C07264=1053.919,247.407,-97.139,172.328,35.943,156.751
C07265=1053.925,247.656,-97.168,172.330,35.946,156.752
C07266=1053.932,247.903,-97.196,172.333,35.950,156.753
C07267=1053.938,248.152,-97.225,172.335,35.954,156.754
C07268=1053.944,248.400,-97.254,172.337,35.957,156.754
C07269=1053.950,248.641,-97.282,172.340,35.960,156.755
C07270=1053.956,248.882,-97.309,172.343,35.964,156.756
C07271=1053.961,249.122,-97.337,172.345,35.967,156.757
C07272=1053.968,249.364,-97.365,172.348,35.970,156.757
C07273=1053.974,249.605,-97.393,172.350,35.974,156.758
C07274=1053.980,249.845,-97.421,172.353,35.977,156.759
C07275=1053.986,250.087,-97.448,172.355,35.980,156.759
C07276=1053.992,250.327,-97.476,172.357,35.984,156.760
C07277=1053.999,250.575,-97.505,172.360,35.987,156.761
C07278=1054.005,250.824,-97.533,172.362,35.991,156.761
C07279=1054.011,251.072,-97.563,172.364,35.994,156.762
C07280=1054.017,251.320,-97.592,172.367,35.998,156.763
C07281=1054.023,251.569,-97.620,172.369,36.001,156.764
C07282=1054.029,251.817,-97.649,172.372,36.005,156.764
C07283=1054.036,252.065,-97.678,172.374,36.008,156.765
C07284=1054.043,252.313,-97.706,172.377,36.012,156.766
C07285=1054.049,252.561,-97.735,172.380,36.015,156.766
C07286=1054.055,252.810,-97.764,172.382,36.018,156.767
C07287=1054.061,253.058,-97.793,172.384,36.022,156.768
C07288=1054.067,253.306,-97.822,172.387,36.025,156.769
C07289=1054.074,253.554,-97.851,172.389,36.029,156.769
C07290=1054.080,253.803,-97.880,172.392,36.033,156.770
C07291=1054.086,254.052,-97.909,172.395,36.036,156.771
C07292=1054.093,254.300,-97.938,172.397,36.039,156.771
C07293=1054.100,254.548,-97.966,172.400,36.043,156.772
C07294=1054.106,254.796,-97.995,172.402,36.046,156.773
C07295=1054.112,255.044,-98.024,172.404,36.050,156.774
C07296=1054.118,255.292,-98.053,172.407,36.053,156.774
C07297=1054.125,255.540,-98.082,172.410,36.056,156.775
C07298=1054.131,255.789,-98.111,172.413,36.060,156.776
C07299=1054.138,256.037,-98.141,172.415,36.063,156.777
C07300=1054.144,256.286,-98.170,172.417,36.066,156.777
C07301=1054.150,256.534,-98.199,172.420,36.070,156.778
C07302=1054.156,256.782,-98.228,172.423,36.073,156.779
C07303=1054.163,257.030,-98.257,172.425,36.077,156.779
C07304=1054.169,257.278,-98.286,172.428,36.081,156.780
C07305=1054.176,257.527,-98.315,172.430,36.083,156.781
C07306=1054.183,257.775,-98.344,172.433,36.087,156.782
C07307=1054.189,258.023,-98.373,172.436,36.091,156.782
C07308=1054.195,258.271,-98.402,172.438,36.094,156.783
C07309=1054.201,258.519,-98.431,172.441,36.097,156.784
C07310=1054.208,258.768,-98.460,172.443,36.101,156.784
C07311=1054.215,259.016,-98.489,172.445,36.104,156.785
C07312=1054.221,259.264,-98.518,172.449,36.108,156.786
C07313=1054.227,259.512,-98.547,172.451,36.111,156.787
C07314=1054.234,259.761,-98.577,172.454,36.114,156.787
C07315=1054.241,260.009,-98.607,172.456,36.118,156.788
C07316=1054.247,260.257,-98.636,172.459,36.121,156.789
C07317=1054.253,260.505,-98.665,172.462,36.124,156.789
C07318=1054.260,260.754,-98.694,172.464,36.128,156.790
C07319=1054.266,261.002,-98.723,172.467,36.131,156.791
C07320=1054.273,261.249,-98.753,172.470,36.135,156.792
C07321=1054.279,261.498,-98.782,172.472,36.138,156.792
C07322=1054.286,261.746,-98.811,172.475,36.141,156.793
C07323=1054.292,261.995,-98.840,172.477,36.145,156.794
C07324=1054.298,262.243,-98.869,172.481,36.149,156.794
C07325=1054.304,262.456,-98.895,172.483,36.151,156.795
C07326=1054.310,262.670,-98.921,172.485,36.154,156.796
C07327=1054.316,262.884,-98.945,172.487,36.157,156.796
C07328=1054.321,263.098,-98.971,172.490,36.160,156.797
C07329=1054.327,263.312,-98.997,172.491,36.163,156.798
C07330=1054.332,263.525,-99.022,172.494,36.166,156.798
C07331=1054.337,263.740,-99.048,172.496,36.169,156.799
C07332=1054.343,263.953,-99.073,172.498,36.172,156.799
C07333=1054.351,264.254,-99.110,172.502,36.176,156.800
C07334=1054.358,264.554,-99.145,172.505,36.180,156.801
C07335=1054.366,264.855,-99.181,172.509,36.185,156.802
C07336=1054.373,265.155,-99.217,172.511,36.189,156.803
C07337=1054.380,265.403,-99.247,172.515,36.192,156.804
C07338=1054.386,265.651,-99.276,172.517,36.196,156.804
C07339=1054.392,265.899,-99.306,172.519,36.199,156.805
C07340=1054.399,266.148,-99.336,172.522,36.203,156.806
C07341=1054.406,266.396,-99.365,172.525,36.206,156.807
C07342=1054.411,266.644,-99.395,172.528,36.210,156.807
C07343=1054.418,266.892,-99.425,172.530,36.213,156.808
C07344=1054.424,267.140,-99.454,172.533,36.216,156.809
C07345=1054.431,267.389,-99.485,172.536,36.220,156.810
C07346=1054.437,267.636,-99.515,172.538,36.223,156.810
C07347=1054.444,267.885,-99.544,172.542,36.227,156.811
C07348=1054.450,268.133,-99.574,172.544,36.230,156.812
C07349=1054.456,268.381,-99.604,172.546,36.234,156.813
C07350=1054.462,268.629,-99.634,172.550,36.238,156.813
C07351=1054.469,268.877,-99.664,172.552,36.241,156.814
C07352=1054.475,269.126,-99.694,172.555,36.245,156.815
C07353=1054.482,269.374,-99.724,172.558,36.248,156.816
C07354=1054.488,269.622,-99.754,172.560,36.251,156.816
C07355=1054.494,269.869,-99.784,172.563,36.255,156.817
C07356=1054.500,270.118,-99.814,172.566,36.258,156.818
C07357=1054.507,270.366,-99.844,172.569,36.262,156.818
C07358=1054.513,270.614,-99.874,172.571,36.265,156.819
C07359=1054.520,270.862,-99.904,172.575,36.269,156.820
C07360=1054.526,271.110,-99.935,172.577,36.272,156.821
C07361=1054.533,271.359,-99.964,172.579,36.276,156.821
C07362=1054.539,271.606,-99.994,172.583,36.279,156.822
C07363=1054.546,271.855,-100.024,172.585,36.283,156.823
C07364=1054.551,272.102,-100.055,172.588,36.286,156.824
C07365=1054.559,272.351,-100.085,172.591,36.290,156.825
C07366=1054.564,272.598,-100.115,172.594,36.293,156.825
C07367=1054.571,272.847,-100.146,172.597,36.297,156.826
C07368=1054.577,273.094,-100.176,172.599,36.300,156.827
C07369=1054.584,273.343,-100.206,172.602,36.304,156.828
C07370=1054.590,273.591,-100.235,172.605,36.307,156.828
C07371=1054.597,273.840,-100.266,172.608,36.311,156.829
C07372=1054.602,274.088,-100.296,172.610,36.314,156.830
C07373=1054.609,274.336,-100.327,172.613,36.318,156.831
C07374=1054.615,274.584,-100.357,172.616,36.322,156.831
C07375=1054.622,274.831,-100.388,172.619,36.324,156.832
C07376=1054.629,275.079,-100.418,172.622,36.328,156.833
C07377=1054.635,275.327,-100.449,172.624,36.331,156.833
C07378=1054.641,275.575,-100.479,172.628,36.335,156.834
C07379=1054.647,275.824,-100.510,172.630,36.339,156.835
C07380=1054.654,276.071,-100.540,172.633,36.342,156.836
C07381=1054.660,276.314,-100.569,172.636,36.346,156.836
C07382=1054.666,276.555,-100.599,172.638,36.349,156.837
C07383=1054.672,276.798,-100.629,172.642,36.353,156.838
C07384=1054.679,277.040,-100.659,172.644,36.356,156.839
C07385=1054.685,277.282,-100.689,172.647,36.360,156.839
C07386=1054.691,277.524,-100.719,172.650,36.363,156.840
C07387=1054.697,277.766,-100.748,172.652,36.367,156.841
C07388=1054.703,278.007,-100.778,172.656,36.370,156.842
C07389=1054.710,278.256,-100.808,172.658,36.373,156.842
C07390=1054.716,278.504,-100.839,172.661,36.377,156.843
C07391=1054.723,278.751,-100.870,172.664,36.381,156.844
C07392=1054.729,279.000,-100.901,172.667,36.384,156.845
C07393=1054.735,279.248,-100.931,172.670,36.388,156.846
C07394=1054.742,279.496,-100.961,172.673,36.391,156.846
C07395=1054.749,279.744,-100.993,172.676,36.395,156.847
C07396=1054.755,279.992,-101.023,172.678,36.398,156.848
C07397=1054.761,280.240,-101.054,172.682,36.402,156.849
C07398=1054.767,280.487,-101.085,172.684,36.405,156.849
C07399=1054.774,280.736,-101.116,172.688,36.409,156.850
C07400=1054.780,280.984,-101.147,172.690,36.412,156.851
C07401=1054.786,281.232,-101.178,172.693,36.416,156.852
C07402=1054.793,281.480,-101.209,172.696,36.419,156.852
C07403=1054.799,281.728,-101.240,172.699,36.423,156.853
C07404=1054.805,281.975,-101.271,172.702,36.427,156.854
C07405=1054.812,282.224,-101.301,172.704,36.430,156.855
C07406=1054.818,282.472,-101.333,172.708,36.434,156.856
C07407=1054.824,282.720,-101.363,172.710,36.437,156.856
C07408=1054.831,282.967,-101.395,172.714,36.441,156.857
C07409=1054.837,283.216,-101.425,172.716,36.444,156.858
C07410=1054.844,283.463,-101.456,172.720,36.448,156.859
C07411=1054.850,283.712,-101.487,172.722,36.452,156.859
C07412=1054.857,283.960,-101.519,172.726,36.455,156.860
C07413=1054.863,284.207,-101.549,172.728,36.459,156.861
C07414=1054.869,284.455,-101.580,172.732,36.462,156.862
C07415=1054.876,284.703,-101.612,172.734,36.466,156.862
C07416=1054.882,284.952,-101.643,172.737,36.469,156.863
C07417=1054.889,285.199,-101.674,172.740,36.473,156.864
C07418=1054.895,285.447,-101.705,172.743,36.477,156.865
C07419=1054.902,285.695,-101.736,172.746,36.481,156.866
C07420=1054.908,285.944,-101.768,172.749,36.484,156.866
C07421=1054.914,286.191,-101.799,172.753,36.488,156.867
C07422=1054.920,286.439,-101.830,172.755,36.491,156.868
C07423=1054.927,286.687,-101.861,172.759,36.495,156.869
C07424=1054.934,286.935,-101.892,172.761,36.498,156.869
C07425=1054.940,287.183,-101.924,172.765,36.502,156.870
C07426=1054.946,287.431,-101.954,172.767,36.506,156.871
C07427=1054.953,287.679,-101.986,172.771,36.509,156.872
C07428=1054.960,287.927,-102.017,172.773,36.513,156.873
C07429=1054.966,288.175,-102.049,172.776,36.516,156.873
C07430=1054.973,288.422,-102.080,172.780,36.520,156.874
C07431=1054.978,288.670,-102.112,172.782,36.524,156.875
C07432=1054.985,288.918,-102.143,172.786,36.527,156.876
C07433=1054.992,289.166,-102.174,172.788,36.531,156.877
C07434=1054.998,289.414,-102.205,172.792,36.534,156.877
C07435=1055.004,289.662,-102.237,172.794,36.538,156.878
C07436=1055.011,289.910,-102.269,172.798,36.542,156.879
C07437=1055.017,290.158,-102.300,172.801,36.545,156.880
C07438=1055.024,290.405,-102.332,172.804,36.549,156.881
C07439=1055.030,290.652,-102.363,172.807,36.553,156.881
C07440=1055.037,290.900,-102.394,172.810,36.556,156.882
C07441=1055.042,291.147,-102.426,172.813,36.560,156.883
C07442=1055.049,291.395,-102.458,172.817,36.563,156.884
C07443=1055.056,291.643,-102.490,172.819,36.567,156.885
C07444=1055.062,291.890,-102.521,172.823,36.571,156.885
C07445=1055.068,292.138,-102.553,172.825,36.574,156.886
C07446=1055.075,292.386,-102.584,172.829,36.578,156.887
C07447=1055.082,292.634,-102.616,172.832,36.582,156.888
C07448=1055.088,292.882,-102.648,172.835,36.585,156.889
C07449=1055.095,293.129,-102.680,172.838,36.589,156.889
C07450=1055.101,293.377,-102.711,172.842,36.593,156.890
C07451=1055.107,293.625,-102.743,172.844,36.596,156.891
C07452=1055.114,293.873,-102.775,172.848,36.600,156.892
C07453=1055.120,294.121,-102.806,172.850,36.604,156.893
C07454=1055.127,294.368,-102.838,172.854,36.607,156.893
C07455=1055.133,294.616,-102.870,172.857,36.611,156.894
C07456=1055.139,294.864,-102.902,172.860,36.615,156.895
C07457=1055.146,295.112,-102.933,172.863,36.618,156.896
C07458=1055.152,295.360,-102.966,172.867,36.622,156.897
C07459=1055.159,295.608,-102.998,172.869,36.626,156.898
C07460=1055.165,295.856,-103.030,172.872,36.629,156.898
C07461=1055.172,296.103,-103.062,172.876,36.633,156.899
C07462=1055.178,296.351,-103.094,172.879,36.637,156.900
C07463=1055.185,296.599,-103.126,172.882,36.640,156.901
C07464=1055.191,296.847,-103.158,172.886,36.644,156.902
C07465=1055.197,297.095,-103.190,172.888,36.648,156.903
C07466=1055.204,297.342,-103.222,172.892,36.652,156.903
C07467=1055.210,297.591,-103.254,172.895,36.656,156.904
C07468=1055.216,297.838,-103.287,172.898,36.659,156.905
C07469=1055.222,298.086,-103.319,172.901,36.663,156.906
C07470=1055.229,298.334,-103.352,172.905,36.667,156.907
C07471=1055.236,298.581,-103.384,172.907,36.671,156.908
C07472=1055.242,298.829,-103.416,172.911,36.674,156.908
C07473=1055.248,299.077,-103.449,172.914,36.678,156.909
C07474=1055.254,299.325,-103.481,172.917,36.682,156.910
C07475=1055.261,299.573,-103.513,172.920,36.686,156.911
C07476=1055.267,299.820,-103.545,172.924,36.690,156.912
C07477=1055.273,300.068,-103.577,172.926,36.693,156.913
C07478=1055.280,300.316,-103.610,172.930,36.697,156.913
C07479=1055.286,300.564,-103.643,172.933,36.701,156.914
C07480=1055.293,300.811,-103.674,172.937,36.705,156.915
C07481=1055.299,301.059,-103.707,172.939,36.709,156.916
C07482=1055.305,301.307,-103.740,172.943,36.712,156.917
C07483=1055.311,301.555,-103.772,172.946,36.717,156.918
C07484=1055.317,301.802,-103.805,172.950,36.720,156.918
C07485=1055.324,302.050,-103.837,172.953,36.724,156.919
C07486=1055.331,302.298,-103.870,172.956,36.728,156.920
C07487=1055.338,302.546,-103.903,172.960,36.731,156.921
C07488=1055.344,302.794,-103.935,172.963,36.736,156.922
C07489=1055.350,303.041,-103.967,172.966,36.739,156.923
C07490=1055.356,303.289,-104.000,172.969,36.743,156.924
C07491=1055.363,303.537,-104.033,172.973,36.747,156.924
C07492=1055.370,303.784,-104.065,172.976,36.751,156.925
C07493=1055.376,304.047,-104.100,172.979,36.755,156.926
C07494=1055.383,304.310,-104.134,172.982,36.759,156.927
C07495=1055.390,304.573,-104.169,172.986,36.763,156.928
C07496=1055.396,304.836,-104.204,172.990,36.767,156.929
C07497=1055.404,305.084,-104.236,172.993,36.771,156.930
C07498=1055.410,305.332,-104.269,172.997,36.775,156.931
C07499=1055.417,305.580,-104.302,173.000,36.778,156.931
C07500=1055.423,305.827,-104.334,173.004,36.782,156.932
C07501=1055.429,306.075,-104.367,173.006,36.786,156.933
C07502=1055.436,306.323,-104.400,173.010,36.790,156.934
C07503=1055.442,306.571,-104.433,173.013,36.794,156.935
C07504=1055.449,306.818,-104.466,173.017,36.798,156.936
C07505=1055.456,307.065,-104.499,173.020,36.801,156.937
C07506=1055.463,307.313,-104.532,173.023,36.805,156.938
C07507=1055.469,307.561,-104.564,173.027,36.809,156.938
C07508=1055.475,307.808,-104.597,173.030,36.813,156.939
C07509=1055.482,308.057,-104.630,173.034,36.817,156.940
C07510=1055.489,308.304,-104.663,173.037,36.821,156.941
C07511=1055.495,308.552,-104.696,173.041,36.825,156.942
C07512=1055.502,308.800,-104.729,173.044,36.828,156.943
C07513=1055.508,309.047,-104.762,173.047,36.832,156.944
C07514=1055.515,309.294,-104.795,173.051,36.836,156.945
C07515=1055.522,309.543,-104.828,173.054,36.840,156.945
C07516=1055.529,309.790,-104.860,173.058,36.844,156.946
C07517=1055.535,310.037,-104.894,173.061,36.848,156.947
C07518=1055.542,310.286,-104.927,173.065,36.852,156.948
C07519=1055.548,310.533,-104.960,173.068,36.855,156.949
C07520=1055.555,310.781,-104.993,173.071,36.859,156.950
C07521=1055.562,311.028,-105.026,173.074,36.863,156.951
C07522=1055.569,311.277,-105.059,173.078,36.867,156.952
C07523=1055.575,311.524,-105.092,173.082,36.871,156.952
C07524=1055.582,311.771,-105.126,173.085,36.875,156.953
C07525=1055.589,312.020,-105.159,173.089,36.879,156.954
C07526=1055.595,312.267,-105.192,173.092,36.883,156.955
C07527=1055.602,312.515,-105.225,173.096,36.886,156.956
C07528=1055.608,312.762,-105.258,173.099,36.890,156.957
C07529=1055.616,313.010,-105.292,173.103,36.894,156.958
C07530=1055.622,313.258,-105.325,173.107,36.898,156.959
C07531=1055.629,313.505,-105.358,173.109,36.902,156.959
C07532=1055.635,313.753,-105.391,173.113,36.906,156.960
C07533=1055.642,314.001,-105.426,173.116,36.910,156.961
C07534=1055.648,314.248,-105.459,173.120,36.914,156.962
C07535=1055.655,314.497,-105.493,173.124,36.918,156.963
C07536=1055.661,314.743,-105.526,173.127,36.922,156.964
C07537=1055.667,314.991,-105.560,173.131,36.926,156.965
C07538=1055.674,315.239,-105.593,173.134,36.930,156.966
C07539=1055.681,315.486,-105.627,173.138,36.934,156.967
C07540=1055.687,315.734,-105.661,173.142,36.939,156.968
C07541=1055.693,315.982,-105.694,173.144,36.943,156.969
C07542=1055.700,316.230,-105.728,173.148,36.947,156.970
C07543=1055.706,316.477,-105.762,173.151,36.951,156.970
C07544=1055.713,316.725,-105.796,173.155,36.955,156.971
C07545=1055.719,316.972,-105.829,173.159,36.959,156.972
C07546=1055.726,317.220,-105.863,173.162,36.963,156.973
C07547=1055.732,317.467,-105.897,173.166,36.967,156.974
C07548=1055.739,317.715,-105.931,173.170,36.971,156.975
C07549=1055.745,317.982,-105.968,173.173,36.975,156.976
C07550=1055.752,318.249,-106.004,173.177,36.980,156.977
C07551=1055.759,318.516,-106.041,173.182,36.984,156.978
C07552=1055.767,318.784,-106.078,173.185,36.989,156.979
C07553=1055.773,319.031,-106.111,173.189,36.993,156.980
C07554=1055.780,319.279,-106.146,173.192,36.997,156.981
C07555=1055.786,319.527,-106.179,173.196,37.001,156.982
C07556=1055.792,319.774,-106.213,173.200,37.005,156.983
C07557=1055.800,320.022,-106.247,173.203,37.009,156.984
C07558=1055.805,320.269,-106.281,173.207,37.013,156.985
C07559=1055.813,320.517,-106.315,173.211,37.017,156.986
C07560=1055.819,320.764,-106.350,173.214,37.021,156.987
C07561=1055.826,321.011,-106.383,173.218,37.026,156.988
C07562=1055.832,321.259,-106.418,173.221,37.030,156.989
C07563=1055.839,321.507,-106.452,173.225,37.034,156.990
C07564=1055.845,321.754,-106.486,173.229,37.038,156.990
C07565=1055.852,322.002,-106.520,173.232,37.042,156.992
C07566=1055.859,322.250,-106.554,173.236,37.046,156.992
C07567=1055.866,322.498,-106.588,173.240,37.050,156.993
C07568=1055.872,322.745,-106.622,173.243,37.054,156.994
C07569=1055.879,322.992,-106.657,173.247,37.059,156.995
C07570=1055.885,323.240,-106.691,173.251,37.063,156.996
C07571=1055.893,323.488,-106.725,173.254,37.067,156.997
C07572=1055.898,323.735,-106.759,173.258,37.071,156.998
C07573=1055.906,323.983,-106.793,173.262,37.075,156.999
C07574=1055.912,324.230,-106.828,173.265,37.079,157.000
C07575=1055.919,324.478,-106.862,173.269,37.084,157.001
C07576=1055.926,324.726,-106.896,173.272,37.088,157.002
C07577=1055.932,324.972,-106.931,173.276,37.092,157.003
C07578=1055.939,325.220,-106.965,173.280,37.096,157.004
C07579=1055.946,325.468,-106.999,173.284,37.100,157.005
C07580=1055.953,325.715,-107.034,173.288,37.105,157.006
C07581=1055.960,325.963,-107.068,173.292,37.109,157.007
C07582=1055.966,326.211,-107.103,173.295,37.113,157.008
C07583=1055.973,326.458,-107.138,173.299,37.117,157.009
C07584=1055.980,326.705,-107.171,173.303,37.121,157.010
C07585=1055.987,326.953,-107.206,173.306,37.126,157.011
C07586=1055.993,327.201,-107.241,173.310,37.130,157.012
C07587=1056.000,327.448,-107.275,173.314,37.134,157.013
C07588=1056.007,327.696,-107.310,173.318,37.138,157.014
C07589=1056.014,327.943,-107.344,173.322,37.142,157.015
C07590=1056.021,328.191,-107.379,173.326,37.147,157.016
C07591=1056.028,328.438,-107.414,173.329,37.151,157.017
C07592=1056.035,328.686,-107.448,173.333,37.155,157.018
C07593=1056.042,328.933,-107.483,173.337,37.159,157.019
C07594=1056.048,329.181,-107.518,173.341,37.164,157.020
C07595=1056.056,329.428,-107.552,173.345,37.168,157.021
C07596=1056.062,329.676,-107.587,173.349,37.172,157.022
C07597=1056.069,329.924,-107.621,173.353,37.176,157.023
C07598=1056.076,330.171,-107.657,173.356,37.181,157.024
C07599=1056.082,330.418,-107.692,173.360,37.185,157.025
C07600=1056.089,330.666,-107.727,173.364,37.189,157.026
C07601=1056.096,330.914,-107.761,173.368,37.194,157.027
C07602=1056.102,331.161,-107.796,173.372,37.198,157.028
C07603=1056.109,331.408,-107.831,173.376,37.203,157.029
C07604=1056.116,331.656,-107.867,173.379,37.207,157.030
C07605=1056.123,331.918,-107.903,173.383,37.212,157.031
C07606=1056.130,332.179,-107.941,173.388,37.216,157.032
C07607=1056.137,332.441,-107.977,173.392,37.221,157.033
C07608=1056.144,332.703,-108.015,173.397,37.225,157.034
C07609=1056.151,332.950,-108.050,173.400,37.230,157.035
C07610=1056.158,333.198,-108.086,173.404,37.234,157.036
C07611=1056.165,333.445,-108.121,173.408,37.239,157.037
C07612=1056.172,333.692,-108.156,173.411,37.243,157.038
C07613=1056.178,333.940,-108.191,173.416,37.248,157.039
C07614=1056.185,334.187,-108.226,173.420,37.252,157.040
C07615=1056.192,334.435,-108.261,173.424,37.256,157.041
C07616=1056.199,334.682,-108.296,173.427,37.261,157.042
C07617=1056.205,334.929,-108.331,173.432,37.265,157.043
C07618=1056.213,335.177,-108.367,173.436,37.270,157.045
C07619=1056.219,335.425,-108.403,173.440,37.274,157.046
C07620=1056.226,335.672,-108.438,173.443,37.279,157.047
C07621=1056.233,335.919,-108.474,173.448,37.283,157.048
C07622=1056.239,336.167,-108.509,173.452,37.288,157.049
C07623=1056.246,336.414,-108.544,173.456,37.292,157.050
C07624=1056.254,336.662,-108.579,173.459,37.297,157.051
C07625=1056.260,336.909,-108.615,173.464,37.301,157.052
C07626=1056.267,337.156,-108.651,173.468,37.306,157.053
C07627=1056.273,337.404,-108.686,173.472,37.310,157.054
C07628=1056.280,337.651,-108.721,173.475,37.315,157.055
C07629=1056.287,337.898,-108.758,173.480,37.319,157.056
C07630=1056.294,338.146,-108.793,173.484,37.324,157.057
C07631=1056.301,338.393,-108.829,173.488,37.329,157.058
C07632=1056.307,338.641,-108.865,173.491,37.333,157.060
C07633=1056.314,338.888,-108.900,173.496,37.338,157.061
C07634=1056.321,339.135,-108.936,173.500,37.342,157.062
C07635=1056.327,339.383,-108.972,173.504,37.347,157.063
C07636=1056.335,339.630,-109.008,173.509,37.352,157.064
C07637=1056.341,339.877,-109.043,173.512,37.356,157.065
C07638=1056.348,340.125,-109.080,173.516,37.361,157.066
C07639=1056.355,340.372,-109.115,173.521,37.365,157.067
C07640=1056.362,340.619,-109.151,173.525,37.370,157.068
C07641=1056.368,340.867,-109.186,173.528,37.375,157.069
C07642=1056.376,341.114,-109.223,173.533,37.379,157.070
C07643=1056.382,341.361,-109.259,173.537,37.384,157.072
C07644=1056.389,341.609,-109.294,173.541,37.389,157.073
C07645=1056.397,341.856,-109.330,173.546,37.393,157.074
C07646=1056.403,342.103,-109.367,173.549,37.398,157.075
C07647=1056.410,342.351,-109.402,173.553,37.403,157.076
C07648=1056.417,342.598,-109.438,173.558,37.407,157.077
C07649=1056.424,342.845,-109.475,173.562,37.412,157.078
C07650=1056.431,343.093,-109.510,173.567,37.417,157.079
C07651=1056.437,343.340,-109.547,173.570,37.421,157.081
C07652=1056.444,343.587,-109.583,173.574,37.426,157.082
C07653=1056.451,343.835,-109.619,173.579,37.431,157.083
C07654=1056.458,344.082,-109.656,173.583,37.436,157.084
C07655=1056.465,344.329,-109.692,173.587,37.440,157.085
C07656=1056.472,344.576,-109.728,173.592,37.445,157.086
C07657=1056.479,344.824,-109.764,173.595,37.450,157.087
C07658=1056.485,345.071,-109.800,173.600,37.455,157.089
C07659=1056.492,345.318,-109.837,173.604,37.459,157.090
C07660=1056.499,345.566,-109.873,173.608,37.464,157.091
C07661=1056.506,345.823,-109.911,173.613,37.469,157.092
C07662=1056.514,346.080,-109.949,173.618,37.474,157.093
C07663=1056.520,346.338,-109.987,173.622,37.479,157.094
C07664=1056.528,346.596,-110.025,173.626,37.484,157.096
C07665=1056.535,346.843,-110.061,173.630,37.489,157.097
C07666=1056.542,347.091,-110.098,173.635,37.494,157.098
C07667=1056.548,347.337,-110.135,173.639,37.499,157.099
C07668=1056.556,347.584,-110.171,173.644,37.504,157.100
C07669=1056.563,347.832,-110.208,173.648,37.508,157.101
C07670=1056.569,348.079,-110.244,173.652,37.513,157.103
C07671=1056.577,348.327,-110.281,173.656,37.518,157.104
C07672=1056.584,348.573,-110.318,173.660,37.523,157.105
C07673=1056.590,348.821,-110.355,173.665,37.528,157.106
C07674=1056.597,349.068,-110.391,173.669,37.533,157.107
C07675=1056.605,349.315,-110.427,173.674,37.538,157.109
C07676=1056.611,349.562,-110.464,173.678,37.543,157.110
C07677=1056.618,349.810,-110.501,173.683,37.548,157.111
C07678=1056.625,350.057,-110.538,173.687,37.553,157.112
C07679=1056.632,350.303,-110.575,173.692,37.558,157.113
C07680=1056.639,350.551,-110.611,173.695,37.563,157.115
C07681=1056.647,350.798,-110.649,173.700,37.568,157.116
C07682=1056.653,351.045,-110.685,173.704,37.572,157.117
C07683=1056.660,351.293,-110.722,173.709,37.577,157.118
C07684=1056.668,351.540,-110.759,173.713,37.583,157.119
C07685=1056.674,351.787,-110.796,173.718,37.588,157.121
C07686=1056.681,352.034,-110.833,173.723,37.593,157.122
C07687=1056.689,352.281,-110.871,173.727,37.598,157.123
C07688=1056.695,352.528,-110.907,173.732,37.603,157.124
C07689=1056.702,352.776,-110.945,173.736,37.608,157.126
C07690=1056.709,353.023,-110.981,173.740,37.613,157.127
C07691=1056.716,353.270,-111.019,173.744,37.618,157.128
C07692=1056.723,353.517,-111.056,173.749,37.623,157.129
C07693=1056.730,353.764,-111.094,173.753,37.628,157.131
C07694=1056.737,354.012,-111.131,173.758,37.633,157.132
C07695=1056.744,354.258,-111.168,173.763,37.638,157.133
C07696=1056.751,354.505,-111.205,173.767,37.643,157.134
C07697=1056.758,354.752,-111.243,173.772,37.649,157.136
C07698=1056.765,355.000,-111.280,173.776,37.654,157.137
C07699=1056.772,355.247,-111.317,173.781,37.659,157.138
C07700=1056.779,355.494,-111.354,173.786,37.664,157.139
C07701=1056.786,355.741,-111.392,173.790,37.669,157.141
C07702=1056.794,355.988,-111.429,173.795,37.674,157.142
C07703=1056.801,356.235,-111.467,173.799,37.680,157.143
C07704=1056.808,356.482,-111.504,173.804,37.685,157.144
C07705=1056.815,356.729,-111.541,173.809,37.689,157.146
C07706=1056.822,356.976,-111.579,173.813,37.695,157.147
C07707=1056.829,357.223,-111.617,173.818,37.700,157.148
C07708=1056.837,357.470,-111.654,173.823,37.705,157.149
C07709=1056.844,357.717,-111.692,173.827,37.710,157.151
C07710=1056.850,357.965,-111.730,173.831,37.715,157.152
C07711=1056.858,358.212,-111.767,173.837,37.721,157.153
C07712=1056.865,358.459,-111.805,173.841,37.726,157.155
C07713=1056.872,358.706,-111.842,173.845,37.731,157.156
C07714=1056.879,358.953,-111.879,173.851,37.737,157.157
C07715=1056.885,359.200,-111.918,173.854,37.742,157.158
C07716=1056.893,359.447,-111.956,173.860,37.747,157.160
C07717=1056.900,359.709,-111.996,173.865,37.753,157.161
C07718=1056.908,359.971,-112.036,173.870,37.759,157.163
C07719=1056.916,360.234,-112.076,173.875,37.765,157.164
C07720=1056.923,360.497,-112.117,173.880,37.770,157.165
C07721=1056.931,360.744,-112.155,173.884,37.776,157.167
C07722=1056.938,360.991,-112.192,173.889,37.781,157.168
C07723=1056.945,361.237,-112.231,173.894,37.787,157.169
C07724=1056.952,361.485,-112.269,173.899,37.791,157.171
C07725=1056.959,361.732,-112.306,173.903,37.797,157.172
C07726=1056.967,361.979,-112.345,173.908,37.802,157.173
C07727=1056.974,362.226,-112.382,173.913,37.808,157.175
C07728=1056.981,362.473,-112.421,173.918,37.813,157.176
C07729=1056.988,362.720,-112.458,173.922,37.819,157.178
C07730=1056.996,362.966,-112.497,173.927,37.824,157.179
C07731=1057.002,363.213,-112.535,173.932,37.830,157.180
C07732=1057.010,363.460,-112.573,173.937,37.835,157.182
C07733=1057.017,363.707,-112.611,173.941,37.841,157.183
C07734=1057.024,363.954,-112.649,173.946,37.846,157.184
C07735=1057.030,364.201,-112.688,173.952,37.852,157.186
C07736=1057.038,364.447,-112.726,173.957,37.857,157.187
C07737=1057.045,364.695,-112.766,173.961,37.863,157.188
C07738=1057.053,364.942,-112.803,173.966,37.868,157.190
C07739=1057.059,365.189,-112.842,173.971,37.874,157.191
C07740=1057.067,365.435,-112.880,173.976,37.880,157.193
C07741=1057.074,365.682,-112.919,173.981,37.885,157.194
C07742=1057.081,365.929,-112.957,173.986,37.891,157.195
C07743=1057.088,366.176,-112.996,173.990,37.897,157.197
C07744=1057.095,366.424,-113.035,173.995,37.902,157.198
C07745=1057.103,366.670,-113.073,174.000,37.908,157.200
C07746=1057.110,366.917,-113.112,174.006,37.914,157.201
C07747=1057.117,367.164,-113.150,174.011,37.919,157.203
C07748=1057.124,367.410,-113.189,174.016,37.925,157.204
C07749=1057.131,367.658,-113.228,174.020,37.931,157.205
C07750=1057.139,367.904,-113.266,174.025,37.936,157.207
C07751=1057.146,368.151,-113.305,174.030,37.942,157.208
C07752=1057.154,368.398,-113.344,174.035,37.948,157.210
C07753=1057.161,368.645,-113.383,174.041,37.954,157.211
C07754=1057.168,368.892,-113.422,174.046,37.959,157.213
C07755=1057.175,369.138,-113.460,174.051,37.965,157.214
C07756=1057.183,369.386,-113.500,174.056,37.971,157.216
C07757=1057.190,369.632,-113.538,174.060,37.977,157.217
C07758=1057.198,369.878,-113.577,174.065,37.982,157.218
C07759=1057.205,370.126,-113.617,174.070,37.988,157.220
C07760=1057.212,370.372,-113.655,174.076,37.994,157.221
C07761=1057.220,370.620,-113.694,174.081,38.000,157.223
C07762=1057.227,370.866,-113.734,174.086,38.006,157.224
C07763=1057.235,371.113,-113.772,174.091,38.012,157.226
C07764=1057.242,371.359,-113.812,174.096,38.017,157.227
C07765=1057.249,371.606,-113.851,174.101,38.023,157.229
C07766=1057.257,371.854,-113.889,174.107,38.029,157.230
C07767=1057.264,372.100,-113.929,174.112,38.035,157.232
C07768=1057.272,372.347,-113.968,174.117,38.041,157.233
C07769=1057.279,372.593,-114.007,174.122,38.047,157.235
C07770=1057.286,372.840,-114.046,174.128,38.053,157.236
C07771=1057.293,373.087,-114.086,174.133,38.059,157.238
C07772=1057.301,373.333,-114.126,174.138,38.065,157.239
C07773=1057.309,373.615,-114.170,174.143,38.072,157.241
C07774=1057.317,373.896,-114.215,174.150,38.079,157.243
C07775=1057.327,374.177,-114.260,174.155,38.086,157.245
C07776=1057.334,374.458,-114.305,174.162,38.092,157.246
C07777=1057.342,374.705,-114.345,174.167,38.099,157.248
C07778=1057.349,374.951,-114.385,174.172,38.105,157.249
C07779=1057.356,375.198,-114.424,174.177,38.111,157.251
C07780=1057.364,375.444,-114.464,174.183,38.117,157.253
C07781=1057.371,375.691,-114.503,174.188,38.123,157.254
C07782=1057.378,375.938,-114.543,174.193,38.129,157.256
C07783=1057.386,376.185,-114.583,174.198,38.135,157.257
C07784=1057.394,376.431,-114.623,174.204,38.141,157.259
C07785=1057.401,376.678,-114.662,174.209,38.148,157.260
C07786=1057.408,376.925,-114.702,174.214,38.154,157.262
C07787=1057.416,377.172,-114.742,174.221,38.160,157.264
C07788=1057.423,377.418,-114.782,174.226,38.166,157.265
C07789=1057.431,377.665,-114.821,174.231,38.172,157.267
C07790=1057.439,377.912,-114.861,174.237,38.179,157.268
C07791=1057.446,378.158,-114.901,174.242,38.185,157.270
C07792=1057.454,378.404,-114.942,174.247,38.191,157.272
C07793=1057.462,378.651,-114.981,174.253,38.198,157.273
C07794=1057.469,378.897,-115.021,174.258,38.204,157.275
C07795=1057.476,379.144,-115.061,174.263,38.210,157.276
C07796=1057.484,379.391,-115.101,174.269,38.216,157.278
C07797=1057.492,379.637,-115.142,174.275,38.222,157.280
C07798=1057.499,379.883,-115.181,174.280,38.229,157.281
C07799=1057.507,380.130,-115.221,174.285,38.235,157.283
C07800=1057.515,380.377,-115.261,174.291,38.241,157.284
C07801=1057.523,380.624,-115.302,174.296,38.248,157.286
C07802=1057.530,380.870,-115.341,174.303,38.254,157.288
C07803=1057.537,381.116,-115.382,174.308,38.261,157.290
C07804=1057.545,381.363,-115.422,174.313,38.267,157.291
C07805=1057.553,381.609,-115.463,174.319,38.274,157.293
C07806=1057.560,381.857,-115.503,174.324,38.280,157.295
C07807=1057.568,382.103,-115.544,174.331,38.287,157.296
C07808=1057.575,382.349,-115.585,174.336,38.293,157.298
C07809=1057.582,382.596,-115.625,174.341,38.300,157.300
C07810=1057.590,382.842,-115.665,174.347,38.306,157.301
C07811=1057.598,383.089,-115.707,174.352,38.313,157.303
C07812=1057.605,383.336,-115.747,174.359,38.320,157.305
C07813=1057.613,383.582,-115.787,174.364,38.326,157.306
C07814=1057.621,383.828,-115.828,174.370,38.333,157.308
C07815=1057.629,384.075,-115.869,174.375,38.340,157.310
C07816=1057.636,384.322,-115.910,174.381,38.346,157.312
C07817=1057.644,384.568,-115.950,174.387,38.353,157.313
C07818=1057.651,384.814,-115.991,174.392,38.360,157.315
C07819=1057.658,385.060,-116.032,174.399,38.366,157.317
C07820=1057.667,385.307,-116.073,174.404,38.373,157.319
C07821=1057.674,385.553,-116.113,174.410,38.379,157.320
C07822=1057.682,385.800,-116.155,174.416,38.386,157.322
C07823=1057.690,386.047,-116.195,174.422,38.393,157.324
C07824=1057.698,386.293,-116.236,174.427,38.400,157.326
C07825=1057.706,386.539,-116.277,174.434,38.406,157.327
C07826=1057.713,386.786,-116.318,174.439,38.413,157.329
C07827=1057.721,387.032,-116.359,174.445,38.420,157.331
C07828=1057.729,387.279,-116.400,174.451,38.427,157.333
C07829=1057.738,387.591,-116.452,174.458,38.435,157.335
C07830=1057.749,387.903,-116.504,174.466,38.444,157.337
C07831=1057.759,388.216,-116.556,174.473,38.453,157.340
C07832=1057.768,388.529,-116.608,174.481,38.462,157.342
C07833=1057.777,388.775,-116.650,174.487,38.469,157.344
C07834=1057.784,389.021,-116.691,174.493,38.475,157.345
C07835=1057.792,389.267,-116.732,174.499,38.482,157.347
C07836=1057.801,389.514,-116.773,174.505,38.489,157.349
C07837=1057.808,389.760,-116.815,174.511,38.496,157.351
C07838=1057.816,390.006,-116.857,174.516,38.503,157.353
C07839=1057.824,390.253,-116.897,174.523,38.510,157.355
C07840=1057.832,390.499,-116.940,174.529,38.517,157.356
C07841=1057.839,390.746,-116.981,174.535,38.524,157.358
C07842=1057.848,390.992,-117.022,174.541,38.531,157.360
C07843=1057.855,391.238,-117.063,174.547,38.539,157.362
C07844=1057.863,391.485,-117.106,174.553,38.546,157.364
C07845=1057.871,391.730,-117.147,174.560,38.552,157.366
C07846=1057.879,391.977,-117.188,174.565,38.560,157.368
C07847=1057.887,392.224,-117.231,174.572,38.567,157.370
C07848=1057.894,392.470,-117.272,174.578,38.574,157.372
C07849=1057.903,392.715,-117.314,174.584,38.581,157.373
C07850=1057.911,392.962,-117.356,174.590,38.589,157.375
C07851=1057.918,393.209,-117.397,174.597,38.596,157.377
C07852=1057.926,393.455,-117.440,174.602,38.603,157.379
C07853=1057.934,393.701,-117.482,174.609,38.610,157.381
C07854=1057.942,393.947,-117.524,174.615,38.618,157.383
C07855=1057.951,394.194,-117.565,174.621,38.625,157.385
C07856=1057.958,394.440,-117.607,174.628,38.632,157.387
C07857=1057.966,394.686,-117.650,174.634,38.640,157.389
C07858=1057.974,394.932,-117.692,174.641,38.647,157.391
C07859=1057.982,395.179,-117.734,174.646,38.654,157.393
C07860=1057.990,395.424,-117.776,174.653,38.662,157.395
C07861=1057.998,395.671,-117.819,174.660,38.669,157.397
C07862=1058.006,395.917,-117.861,174.666,38.677,157.399
C07863=1058.014,396.164,-117.903,174.672,38.684,157.401
C07864=1058.022,396.410,-117.945,174.679,38.691,157.403
C07865=1058.030,396.656,-117.988,174.685,38.699,157.405
C07866=1058.038,396.902,-118.030,174.692,38.706,157.407
C07867=1058.047,397.148,-118.072,174.697,38.714,157.409
C07868=1058.054,397.394,-118.115,174.704,38.722,157.411
C07869=1058.063,397.641,-118.158,174.711,38.729,157.413
C07870=1058.070,397.887,-118.200,174.717,38.737,157.415
C07871=1058.079,398.133,-118.243,174.724,38.745,157.417
C07872=1058.087,398.380,-118.285,174.730,38.752,157.419
C07873=1058.095,398.625,-118.328,174.737,38.760,157.421
C07874=1058.103,398.871,-118.371,174.743,38.767,157.423
C07875=1058.112,399.118,-118.413,174.750,38.775,157.425
C07876=1058.119,399.363,-118.456,174.757,38.783,157.428
C07877=1058.127,399.610,-118.498,174.763,38.791,157.430
C07878=1058.135,399.856,-118.541,174.770,38.799,157.432
C07879=1058.144,400.102,-118.585,174.777,38.807,157.434
C07880=1058.152,400.348,-118.628,174.783,38.814,157.436
C07881=1058.160,400.594,-118.669,174.790,38.822,157.438
C07882=1058.168,400.840,-118.713,174.796,38.830,157.440
C07883=1058.176,401.087,-118.756,174.803,38.838,157.442
C07884=1058.185,401.333,-118.799,174.810,38.846,157.445
C07885=1058.196,401.663,-118.856,174.819,38.856,157.447
C07886=1058.207,401.992,-118.914,174.828,38.867,157.450
C07887=1058.218,402.323,-118.972,174.837,38.877,157.453
C07888=1058.229,402.652,-119.030,174.846,38.888,157.456
C07889=1058.237,402.898,-119.074,174.853,38.896,157.458
C07890=1058.245,403.144,-119.117,174.860,38.904,157.460
C07891=1058.254,403.390,-119.160,174.866,38.912,157.463
C07892=1058.262,403.637,-119.203,174.873,38.920,157.465
C07893=1058.270,403.882,-119.247,174.881,38.929,157.467
C07894=1058.279,404.128,-119.290,174.887,38.936,157.469
C07895=1058.287,404.374,-119.334,174.895,38.945,157.472
C07896=1058.295,404.621,-119.377,174.902,38.953,157.474
C07897=1058.304,404.867,-119.421,174.909,38.961,157.476
C07898=1058.312,405.113,-119.464,174.916,38.969,157.478
C07899=1058.320,405.359,-119.509,174.923,38.977,157.481
C07900=1058.329,405.605,-119.552,174.930,38.986,157.483
C07901=1058.337,405.851,-119.595,174.937,38.994,157.485
C07902=1058.345,406.097,-119.639,174.944,39.003,157.487
C07903=1058.354,406.342,-119.683,174.951,39.011,157.490
C07904=1058.361,406.589,-119.727,174.958,39.019,157.492
C07905=1058.371,406.835,-119.771,174.965,39.027,157.494
C07906=1058.378,407.081,-119.815,174.972,39.036,157.497
C07907=1058.387,407.327,-119.859,174.980,39.045,157.499
C07908=1058.395,407.572,-119.903,174.987,39.053,157.501
C07909=1058.404,407.819,-119.948,174.994,39.061,157.504
C07910=1058.413,408.065,-119.991,175.001,39.070,157.506
C07911=1058.421,408.311,-120.035,175.008,39.078,157.508
C07912=1058.429,408.556,-120.079,175.016,39.087,157.511
C07913=1058.438,408.803,-120.123,175.023,39.095,157.513
C07914=1058.446,409.048,-120.168,175.030,39.104,157.515
C07915=1058.454,409.294,-120.212,175.037,39.113,157.518
C07916=1058.464,409.540,-120.256,175.045,39.121,157.520
C07917=1058.472,409.786,-120.300,175.053,39.130,157.523
C07918=1058.480,410.032,-120.345,175.060,39.139,157.525
C07919=1058.489,410.278,-120.389,175.067,39.147,157.527
C07920=1058.498,410.524,-120.434,175.074,39.156,157.530
C07921=1058.506,410.770,-120.478,175.083,39.165,157.532
C07922=1058.514,411.015,-120.523,175.090,39.173,157.535
C07923=1058.524,411.261,-120.567,175.097,39.182,157.537
C07924=1058.532,411.508,-120.612,175.105,39.191,157.540
C07925=1058.540,411.753,-120.656,175.112,39.200,157.542
C07926=1058.550,411.999,-120.701,175.120,39.209,157.545
C07927=1058.558,412.245,-120.745,175.128,39.218,157.547
C07928=1058.567,412.491,-120.790,175.135,39.227,157.550
C07929=1058.575,412.736,-120.835,175.143,39.235,157.552
C07930=1058.585,412.982,-120.879,175.151,39.244,157.555
C07931=1058.594,413.228,-120.925,175.158,39.254,157.557
C07932=1058.602,413.474,-120.969,175.166,39.262,157.560
C07933=1058.611,413.720,-121.014,175.174,39.271,157.562
C07934=1058.619,413.966,-121.059,175.181,39.281,157.565
C07935=1058.628,414.212,-121.104,175.190,39.289,157.567
C07936=1058.637,414.457,-121.150,175.197,39.299,157.570
C07937=1058.646,414.703,-121.195,175.205,39.308,157.573
C07938=1058.655,414.949,-121.240,175.213,39.317,157.575
C07939=1058.663,415.195,-121.285,175.221,39.326,157.578
C07940=1058.672,415.440,-121.330,175.229,39.336,157.580
C07941=1058.679,415.655,-121.370,175.235,39.344,157.583
C07942=1058.687,415.870,-121.409,175.242,39.352,157.585
C07943=1058.696,416.085,-121.449,175.250,39.360,157.587
C07944=1058.703,416.300,-121.489,175.257,39.368,157.590
C07945=1058.710,416.515,-121.529,175.264,39.376,157.592
C07946=1058.719,416.729,-121.568,175.270,39.384,157.594
C07947=1058.726,416.944,-121.608,175.278,39.393,157.597
C07948=1058.734,417.159,-121.648,175.285,39.401,157.599
C07949=1058.743,417.405,-121.693,175.293,39.410,157.602
C07950=1058.752,417.651,-121.739,175.301,39.420,157.604
C07951=1058.761,417.897,-121.784,175.310,39.429,157.607
C07952=1058.770,418.142,-121.830,175.317,39.439,157.610
C07953=1058.779,418.388,-121.876,175.326,39.448,157.613
C07954=1058.787,418.634,-121.922,175.334,39.458,157.615
C07955=1058.796,418.879,-121.968,175.342,39.467,157.618
C07956=1058.805,419.125,-122.013,175.351,39.477,157.621
C07957=1058.815,419.370,-122.060,175.359,39.487,157.624
C07958=1058.824,419.616,-122.105,175.367,39.496,157.626
C07959=1058.834,419.862,-122.151,175.376,39.506,157.629
C07960=1058.842,420.108,-122.197,175.384,39.516,157.632
C07961=1058.851,420.353,-122.244,175.393,39.526,157.635
C07962=1058.860,420.598,-122.290,175.401,39.535,157.638
C07963=1058.869,420.844,-122.336,175.410,39.545,157.640
C07964=1058.878,421.090,-122.382,175.418,39.555,157.643
C07965=1058.887,421.335,-122.428,175.427,39.565,157.646
C07966=1058.896,421.580,-122.475,175.435,39.575,157.649
C07967=1058.906,421.826,-122.521,175.444,39.585,157.652
C07968=1058.915,422.071,-122.567,175.452,39.595,157.655
C07969=1058.923,422.317,-122.614,175.461,39.605,157.658
C07970=1058.933,422.562,-122.660,175.470,39.615,157.661
C07971=1058.942,422.808,-122.707,175.479,39.625,157.663
C07972=1058.951,423.054,-122.753,175.488,39.635,157.666
C07973=1058.960,423.299,-122.800,175.497,39.645,157.669
C07974=1058.970,423.545,-122.847,175.504,39.656,157.672
C07975=1058.979,423.790,-122.894,175.513,39.666,157.675
C07976=1058.988,424.035,-122.940,175.522,39.676,157.678
C07977=1058.998,424.281,-122.987,175.531,39.686,157.681
C07978=1059.006,424.527,-123.034,175.540,39.697,157.684
C07979=1059.016,424.772,-123.081,175.549,39.707,157.687
C07980=1059.025,425.017,-123.127,175.558,39.717,157.690
C07981=1059.034,425.262,-123.174,175.567,39.727,157.693
C07982=1059.044,425.508,-123.221,175.576,39.737,157.696
C07983=1059.053,425.753,-123.268,175.585,39.748,157.699
C07984=1059.063,425.999,-123.315,175.594,39.758,157.702
C07985=1059.072,426.244,-123.363,175.604,39.769,157.706
C07986=1059.081,426.489,-123.410,175.613,39.779,157.709
C07987=1059.091,426.735,-123.457,175.622,39.790,157.712
C07988=1059.100,426.980,-123.504,175.632,39.801,157.715
C07989=1059.116,427.376,-123.581,175.646,39.818,157.720
C07990=1059.131,427.773,-123.658,175.661,39.835,157.725
C07991=1059.146,428.168,-123.734,175.676,39.853,157.730
C07992=1059.161,428.565,-123.811,175.691,39.870,157.735
C07993=1059.171,428.810,-123.858,175.702,39.880,157.739
C07994=1059.181,429.055,-123.906,175.711,39.892,157.742
C07995=1059.190,429.300,-123.955,175.720,39.902,157.745
C07996=1059.200,429.545,-124.001,175.730,39.913,157.748
C07997=1059.214,429.902,-124.071,175.744,39.929,157.753
C07998=1059.228,430.259,-124.141,175.758,39.945,157.758
C07999=1059.242,430.615,-124.211,175.772,39.961,157.763
C08000=1059.256,430.971,-124.281,175.786,39.977,157.767
C08001=1059.265,431.217,-124.328,175.797,39.989,157.771
C08002=1059.275,431.462,-124.377,175.806,40.000,157.774
C08003=1059.285,431.707,-124.425,175.815,40.011,157.778
C08004=1059.295,431.952,-124.474,175.826,40.022,157.781
C08005=1059.304,432.197,-124.522,175.835,40.034,157.784
C08006=1059.314,432.442,-124.570,175.846,40.045,157.788
C08007=1059.324,432.687,-124.619,175.856,40.056,157.791
C08008=1059.333,432.932,-124.667,175.866,40.067,157.795
C08009=1059.343,433.177,-124.716,175.876,40.079,157.798
C08010=1059.353,433.422,-124.764,175.886,40.091,157.802
C08011=1059.363,433.667,-124.813,175.896,40.102,157.805
C08012=1059.372,433.912,-124.861,175.906,40.114,157.809
C08013=1059.382,434.157,-124.910,175.917,40.125,157.812
C08014=1059.393,434.403,-124.959,175.927,40.137,157.816
C08015=1059.403,434.647,-125.008,175.937,40.148,157.819
C08016=1059.412,434.892,-125.057,175.948,40.160,157.823
C08017=1059.422,435.137,-125.105,175.958,40.172,157.826
C08018=1059.433,435.382,-125.155,175.969,40.184,157.830
C08019=1059.443,435.627,-125.203,175.979,40.195,157.833
C08020=1059.453,435.871,-125.253,175.990,40.207,157.837
C08021=1059.463,436.117,-125.301,176.000,40.219,157.841
C08022=1059.473,436.361,-125.351,176.011,40.231,157.844
C08023=1059.482,436.607,-125.400,176.021,40.243,157.848
C08024=1059.493,436.852,-125.449,176.032,40.255,157.852
C08025=1059.503,437.096,-125.499,176.043,40.267,157.855
C08026=1059.513,437.342,-125.548,176.053,40.279,157.859
C08027=1059.523,437.586,-125.597,176.064,40.291,157.863
C08028=1059.534,437.831,-125.646,176.075,40.303,157.866
C08029=1059.543,438.076,-125.696,176.086,40.315,157.870
C08030=1059.554,438.321,-125.746,176.097,40.327,157.874
C08031=1059.564,438.565,-125.795,176.108,40.339,157.878
C08032=1059.575,438.810,-125.845,176.119,40.351,157.881
C08033=1059.584,439.055,-125.895,176.130,40.364,157.885
C08034=1059.595,439.299,-125.945,176.141,40.376,157.889
C08035=1059.606,439.545,-125.994,176.152,40.389,157.893
C08036=1059.615,439.789,-126.044,176.163,40.401,157.897
C08037=1059.626,440.034,-126.094,176.174,40.414,157.901
C08038=1059.637,440.279,-126.144,176.185,40.426,157.905
C08039=1059.646,440.523,-126.194,176.198,40.439,157.909
C08040=1059.657,440.768,-126.244,176.209,40.451,157.912
C08041=1059.667,441.013,-126.295,176.220,40.464,157.916
C08042=1059.678,441.258,-126.345,176.231,40.477,157.920
C08043=1059.689,441.502,-126.395,176.243,40.490,157.924
C08044=1059.698,441.746,-126.446,176.255,40.502,157.928
C08045=1059.709,441.991,-126.495,176.266,40.515,157.932
C08046=1059.719,442.236,-126.546,176.278,40.528,157.936
C08047=1059.730,442.480,-126.597,176.289,40.540,157.940
C08048=1059.741,442.725,-126.648,176.301,40.553,157.944
C08049=1059.751,442.969,-126.698,176.313,40.567,157.949
C08050=1059.762,443.214,-126.749,176.324,40.579,157.953
C08051=1059.773,443.459,-126.799,176.337,40.592,157.957
C08052=1059.783,443.703,-126.850,176.348,40.606,157.961
C08053=1059.799,444.048,-126.922,176.366,40.624,157.967
C08054=1059.813,444.392,-126.994,176.382,40.642,157.973
C08055=1059.828,444.737,-127.065,176.399,40.661,157.979
C08056=1059.843,445.082,-127.138,176.417,40.680,157.985
C08057=1059.854,445.326,-127.189,176.429,40.694,157.989
C08058=1059.865,445.571,-127.240,176.441,40.707,157.993
C08059=1059.876,445.816,-127.292,176.454,40.720,157.998
C08060=1059.887,446.059,-127.343,176.466,40.734,158.002
C08061=1059.898,446.304,-127.394,176.479,40.747,158.006
C08062=1059.908,446.549,-127.446,176.491,40.761,158.010
C08063=1059.920,446.793,-127.497,176.503,40.774,158.015
C08064=1059.930,447.037,-127.548,176.516,40.788,158.019
C08065=1059.942,447.280,-127.600,176.529,40.802,158.024
C08066=1059.955,447.523,-127.650,176.542,40.815,158.028
C08067=1059.966,447.767,-127.700,176.554,40.828,158.032
C08068=1059.981,448.012,-127.750,176.567,40.841,158.036
C08069=1059.996,448.256,-127.798,176.581,40.853,158.041
C08070=1060.011,448.500,-127.846,176.593,40.866,158.045
C08071=1060.028,448.745,-127.893,176.606,40.878,158.049
C08072=1060.046,448.990,-127.941,176.620,40.890,158.053
C08073=1060.064,449.234,-127.987,176.632,40.902,158.057
C08074=1060.083,449.480,-128.033,176.646,40.913,158.060
C08075=1060.103,449.725,-128.078,176.660,40.924,158.064
C08076=1060.124,449.970,-128.121,176.673,40.935,158.068
C08077=1059.794,449.982,-128.401,176.668,41.048,158.099
C08078=1059.773,449.738,-128.356,176.654,41.037,158.095
C08079=1059.752,449.492,-128.312,176.641,41.026,158.092
C08080=1059.733,449.247,-128.266,176.628,41.014,158.088
C08081=1059.714,449.001,-128.219,176.614,41.003,158.084
C08082=1059.697,448.756,-128.173,176.601,40.991,158.080
C08083=1059.680,448.512,-128.125,176.587,40.979,158.076
C08084=1059.664,448.268,-128.077,176.575,40.966,158.072
C08085=1059.649,448.024,-128.029,176.561,40.954,158.067
C08086=1059.635,447.779,-127.979,176.548,40.941,158.063
C08087=1059.621,447.535,-127.929,176.536,40.928,158.059
C08088=1059.609,447.291,-127.879,176.523,40.915,158.055
C08089=1059.598,447.049,-127.828,176.510,40.902,158.050
C08090=1059.587,446.804,-127.776,176.497,40.888,158.046
C08091=1059.576,446.560,-127.724,176.484,40.875,158.042
C08092=1059.565,446.316,-127.674,176.472,40.861,158.037
C08093=1059.554,446.071,-127.622,176.459,40.847,158.033
C08094=1059.543,445.827,-127.570,176.447,40.834,158.029
C08095=1059.532,445.583,-127.519,176.434,40.821,158.024
C08096=1059.522,445.338,-127.468,176.422,40.807,158.020
C08097=1059.510,445.094,-127.417,176.409,40.794,158.016
C08098=1059.496,444.768,-127.349,176.393,40.776,158.010
C08099=1059.482,444.443,-127.280,176.377,40.759,158.004
C08100=1059.468,444.117,-127.213,176.361,40.742,157.999
C08101=1059.454,443.792,-127.145,176.345,40.724,157.993
C08102=1059.443,443.548,-127.095,176.333,40.711,157.989
C08103=1059.432,443.304,-127.043,176.321,40.698,157.985
C08104=1059.421,443.059,-126.993,176.309,40.685,157.981
C08105=1059.411,442.814,-126.942,176.297,40.672,157.977
C08106=1059.400,442.570,-126.892,176.285,40.659,157.972
C08107=1059.390,442.325,-126.841,176.274,40.646,157.968
C08108=1059.379,442.081,-126.790,176.261,40.634,157.964
C08109=1059.368,441.836,-126.739,176.250,40.621,157.960
C08110=1059.358,441.591,-126.690,176.239,40.608,157.956
C08111=1059.347,441.346,-126.639,176.226,40.595,157.952
C08112=1059.337,441.102,-126.589,176.215,40.583,157.948
C08113=1059.326,440.858,-126.539,176.204,40.570,157.944
C08114=1059.316,440.613,-126.488,176.192,40.558,157.940
C08115=1059.305,440.368,-126.438,176.181,40.545,157.937
C08116=1059.295,440.123,-126.388,176.169,40.533,157.933
C08117=1059.285,439.879,-126.338,176.158,40.520,157.929
C08118=1059.274,439.634,-126.288,176.147,40.508,157.925
C08119=1059.264,439.389,-126.238,176.136,40.496,157.921
C08120=1059.253,439.144,-126.188,176.124,40.483,157.917
C08121=1059.243,438.900,-126.139,176.113,40.471,157.913
C08122=1059.233,438.655,-126.088,176.102,40.458,157.909
C08123=1059.223,438.410,-126.039,176.091,40.446,157.906
C08124=1059.213,438.165,-125.989,176.080,40.434,157.902
C08125=1059.203,437.921,-125.940,176.069,40.422,157.898
C08126=1059.193,437.675,-125.890,176.058,40.410,157.894
C08127=1059.183,437.431,-125.841,176.047,40.398,157.891
C08128=1059.172,437.186,-125.791,176.036,40.386,157.887
C08129=1059.161,436.941,-125.742,176.025,40.374,157.883
C08130=1059.151,436.696,-125.693,176.015,40.362,157.880
C08131=1059.141,436.451,-125.643,176.004,40.350,157.876
C08132=1059.131,436.207,-125.594,175.993,40.338,157.872
C08133=1059.121,435.962,-125.546,175.983,40.327,157.869
C08134=1059.110,435.717,-125.496,175.972,40.315,157.865
C08135=1059.101,435.471,-125.447,175.962,40.303,157.861
C08136=1059.091,435.227,-125.398,175.951,40.291,157.858
C08137=1059.081,434.981,-125.349,175.940,40.280,157.854
C08138=1059.071,434.737,-125.300,175.930,40.268,157.851
C08139=1059.061,434.492,-125.251,175.920,40.257,157.847
C08140=1059.051,434.247,-125.202,175.909,40.245,157.844
C08141=1059.041,434.001,-125.154,175.899,40.234,157.840
C08142=1059.031,433.757,-125.104,175.889,40.222,157.837
C08143=1059.021,433.512,-125.056,175.878,40.210,157.833
C08144=1059.011,433.267,-125.007,175.869,40.199,157.830
C08145=1059.002,433.022,-124.959,175.858,40.188,157.826
C08146=1058.992,432.777,-124.910,175.848,40.176,157.823
C08147=1058.982,432.532,-124.862,175.838,40.165,157.819
C08148=1058.972,432.287,-124.813,175.828,40.154,157.816
C08149=1058.963,432.042,-124.765,175.818,40.142,157.812
C08150=1058.953,431.797,-124.717,175.808,40.131,157.809
C08151=1058.943,431.552,-124.668,175.798,40.120,157.806
C08152=1058.934,431.307,-124.620,175.788,40.109,157.802
C08153=1058.923,431.062,-124.572,175.778,40.098,157.799
C08154=1058.910,430.703,-124.502,175.764,40.081,157.794
C08155=1058.895,430.344,-124.431,175.750,40.065,157.789
C08156=1058.881,429.987,-124.361,175.735,40.049,157.784
C08157=1058.866,429.627,-124.291,175.721,40.033,157.779
C08158=1058.858,429.382,-124.244,175.711,40.022,157.776
C08159=1058.848,429.138,-124.195,175.701,40.011,157.773
C08160=1058.838,428.892,-124.147,175.692,40.001,157.770
C08161=1058.828,428.647,-124.100,175.682,39.990,157.767
C08162=1058.819,428.402,-124.053,175.673,39.979,157.763
C08163=1058.810,428.156,-124.005,175.664,39.968,157.760
C08164=1058.799,427.911,-123.957,175.653,39.957,157.757
C08165=1058.790,427.666,-123.909,175.644,39.947,157.754
C08166=1058.781,427.421,-123.862,175.635,39.936,157.751
C08167=1058.772,427.175,-123.815,175.626,39.926,157.747
C08168=1058.762,426.930,-123.768,175.617,39.915,157.744
C08169=1058.753,426.685,-123.720,175.607,39.904,157.741
C08170=1058.743,426.439,-123.672,175.597,39.894,157.738
C08171=1058.734,426.194,-123.625,175.588,39.884,157.735
C08172=1058.725,425.948,-123.578,175.579,39.873,157.732
C08173=1058.714,425.703,-123.531,175.570,39.863,157.729
C08174=1058.706,425.458,-123.484,175.561,39.853,157.726
C08175=1058.696,425.212,-123.437,175.552,39.842,157.723
C08176=1058.686,424.968,-123.390,175.543,39.832,157.720
C08177=1058.677,424.721,-123.343,175.534,39.821,157.717
C08178=1058.667,424.477,-123.296,175.525,39.811,157.714
C08179=1058.659,424.231,-123.250,175.516,39.801,157.711
C08180=1058.649,423.985,-123.203,175.507,39.791,157.708
C08181=1058.640,423.740,-123.156,175.498,39.781,157.705
C08182=1058.630,423.495,-123.109,175.489,39.770,157.702
C08183=1058.621,423.249,-123.063,175.480,39.760,157.699
C08184=1058.612,423.004,-123.016,175.472,39.750,157.696
C08185=1058.602,422.758,-122.970,175.463,39.740,157.693
C08186=1058.594,422.513,-122.922,175.454,39.730,157.690
C08187=1058.584,422.268,-122.876,175.445,39.720,157.687
C08188=1058.574,422.022,-122.830,175.436,39.711,157.684
C08189=1058.566,421.776,-122.783,175.427,39.700,157.681
C08190=1058.557,421.531,-122.737,175.419,39.690,157.678
C08191=1058.548,421.286,-122.690,175.410,39.681,157.675
C08192=1058.539,421.040,-122.645,175.402,39.670,157.672
C08193=1058.530,420.795,-122.599,175.393,39.661,157.670
C08194=1058.521,420.548,-122.551,175.385,39.651,157.667
C08195=1058.511,420.303,-122.505,175.376,39.641,157.664
C08196=1058.502,420.058,-122.459,175.367,39.631,157.661
C08197=1058.494,419.812,-122.413,175.359,39.622,157.658
C08198=1058.485,419.567,-122.367,175.351,39.612,157.656
C08199=1058.476,419.321,-122.322,175.342,39.603,157.653
C08200=1058.466,419.076,-122.275,175.333,39.593,157.650
C08201=1058.457,418.830,-122.230,175.326,39.584,157.647
C08202=1058.445,418.502,-122.169,175.314,39.571,157.644
C08203=1058.433,418.175,-122.108,175.303,39.558,157.640
C08204=1058.421,417.849,-122.047,175.292,39.545,157.636
C08205=1058.409,417.521,-121.986,175.281,39.533,157.633
C08206=1058.400,417.275,-121.941,175.273,39.523,157.630
C08207=1058.391,417.030,-121.894,175.265,39.514,157.627
C08208=1058.383,416.785,-121.849,175.257,39.505,157.625
C08209=1058.374,416.539,-121.804,175.249,39.495,157.622
C08210=1058.364,416.283,-121.757,175.240,39.485,157.619
C08211=1058.355,416.027,-121.710,175.231,39.476,157.616
C08212=1058.346,415.771,-121.662,175.224,39.466,157.614
C08213=1058.336,415.516,-121.615,175.215,39.456,157.611
C08214=1058.328,415.269,-121.570,175.207,39.447,157.608
C08215=1058.319,415.024,-121.524,175.199,39.438,157.606
C08216=1058.310,414.778,-121.479,175.192,39.429,157.603
C08217=1058.301,414.533,-121.434,175.183,39.420,157.600
C08218=1058.293,414.286,-121.388,175.176,39.411,157.598
C08219=1058.285,414.041,-121.343,175.167,39.402,157.595
C08220=1058.276,413.795,-121.298,175.160,39.393,157.593
C08221=1058.266,413.549,-121.253,175.152,39.383,157.590
C08222=1058.257,413.304,-121.208,175.144,39.375,157.588
C08223=1058.249,413.058,-121.164,175.136,39.366,157.585
C08224=1058.240,412.812,-121.118,175.129,39.357,157.583
C08225=1058.231,412.566,-121.074,175.121,39.348,157.580
C08226=1058.222,412.321,-121.029,175.113,39.339,157.578
C08227=1058.214,412.074,-120.984,175.106,39.330,157.575
C08228=1058.204,411.828,-120.940,175.097,39.322,157.573
C08229=1058.196,411.583,-120.895,175.090,39.313,157.570
C08230=1058.187,411.337,-120.851,175.083,39.304,157.568
C08231=1058.179,411.091,-120.806,175.075,39.295,157.565
C08232=1058.170,410.845,-120.762,175.067,39.286,157.563
C08233=1058.161,410.600,-120.717,175.060,39.278,157.560
C08234=1058.153,410.353,-120.672,175.052,39.269,157.558
C08235=1058.144,410.108,-120.629,175.045,39.260,157.555
C08236=1058.135,409.861,-120.584,175.038,39.252,157.553
C08237=1058.127,409.615,-120.540,175.029,39.243,157.551
C08238=1058.118,409.370,-120.496,175.022,39.234,157.548
C08239=1058.110,409.124,-120.451,175.015,39.226,157.546
C08240=1058.102,408.878,-120.407,175.008,39.217,157.543
C08241=1058.092,408.632,-120.363,175.001,39.209,157.541
C08242=1058.084,408.386,-120.318,174.993,39.200,157.539
C08243=1058.076,408.140,-120.274,174.986,39.192,157.536
C08244=1058.067,407.894,-120.230,174.979,39.183,157.534
C08245=1058.059,407.648,-120.186,174.972,39.175,157.532
C08246=1058.051,407.402,-120.142,174.964,39.166,157.529
C08247=1058.042,407.157,-120.098,174.956,39.158,157.527
C08248=1058.033,406.910,-120.053,174.949,39.149,157.524
C08249=1058.025,406.664,-120.010,174.942,39.141,157.522
C08250=1058.017,406.418,-119.966,174.935,39.133,157.520
C08251=1058.009,406.173,-119.922,174.928,39.125,157.518
C08252=1058.000,405.927,-119.879,174.920,39.116,157.515
C08253=1057.992,405.681,-119.834,174.913,39.108,157.513
C08254=1057.983,405.434,-119.791,174.906,39.099,157.511
C08255=1057.975,405.188,-119.747,174.899,39.092,157.508
C08256=1057.967,404.942,-119.704,174.893,39.083,157.506
C08257=1057.958,404.696,-119.659,174.886,39.075,157.504
C08258=1057.950,404.450,-119.616,174.879,39.067,157.502
C08259=1057.942,404.204,-119.573,174.872,39.058,157.499
C08260=1057.933,403.959,-119.529,174.865,39.050,157.497
C08261=1057.926,403.712,-119.485,174.858,39.043,157.495
C08262=1057.917,403.466,-119.442,174.851,39.034,157.493
C08263=1057.909,403.220,-119.399,174.844,39.026,157.490
C08264=1057.901,402.974,-119.356,174.837,39.018,157.488
C08265=1057.892,402.728,-119.312,174.830,39.011,157.486
C08266=1057.880,402.396,-119.253,174.821,38.999,157.483
C08267=1057.869,402.065,-119.195,174.811,38.989,157.480
C08268=1057.858,401.732,-119.138,174.802,38.978,157.477
C08269=1057.847,401.401,-119.080,174.793,38.968,157.474
C08270=1057.839,401.154,-119.036,174.786,38.960,157.472
C08271=1057.831,400.908,-118.993,174.780,38.952,157.470
C08272=1057.822,400.662,-118.950,174.773,38.944,157.468
C08273=1057.814,400.417,-118.907,174.766,38.936,157.466
C08274=1057.806,400.170,-118.865,174.759,38.929,157.464
C08275=1057.798,399.924,-118.822,174.752,38.921,157.462
C08276=1057.790,399.678,-118.778,174.746,38.913,157.459
C08277=1057.781,399.432,-118.735,174.739,38.905,157.457
C08278=1057.774,399.186,-118.693,174.732,38.898,157.455
C08279=1057.765,398.940,-118.650,174.726,38.890,157.453
C08280=1057.757,398.694,-118.607,174.720,38.882,157.451
C08281=1057.749,398.447,-118.565,174.713,38.875,157.449
C08282=1057.741,398.202,-118.522,174.706,38.867,157.447
C08283=1057.733,397.955,-118.480,174.700,38.859,157.445
C08284=1057.725,397.709,-118.436,174.693,38.852,157.443
C08285=1057.717,397.463,-118.394,174.686,38.844,157.441
C08286=1057.709,397.217,-118.351,174.681,38.837,157.439
C08287=1057.700,396.970,-118.309,174.674,38.829,157.437
C08288=1057.693,396.724,-118.267,174.667,38.822,157.435
C08289=1057.684,396.478,-118.224,174.661,38.814,157.433
C08290=1057.676,396.231,-118.182,174.654,38.807,157.431
C08291=1057.669,395.985,-118.140,174.648,38.800,157.429
C08292=1057.660,395.739,-118.098,174.642,38.792,157.427
C08293=1057.652,395.494,-118.056,174.635,38.785,157.425
C08294=1057.644,395.247,-118.013,174.628,38.777,157.423
C08295=1057.636,395.001,-117.971,174.622,38.770,157.421
C08296=1057.628,394.754,-117.929,174.616,38.762,157.419
C08297=1057.620,394.508,-117.887,174.610,38.755,157.417
C08298=1057.612,394.262,-117.845,174.603,38.748,157.415
C08299=1057.604,394.016,-117.803,174.596,38.741,157.413
C08300=1057.596,393.769,-117.760,174.591,38.733,157.411
C08301=1057.588,393.523,-117.719,174.584,38.726,157.409
C08302=1057.580,393.277,-117.677,174.578,38.719,157.407
C08303=1057.572,393.031,-117.635,174.571,38.711,157.405
C08304=1057.564,392.785,-117.593,174.566,38.704,157.403
C08305=1057.556,392.538,-117.551,174.559,38.697,157.401
C08306=1057.548,392.292,-117.510,174.553,38.690,157.399
C08307=1057.541,392.046,-117.468,174.547,38.682,157.397
C08308=1057.532,391.799,-117.426,174.541,38.675,157.396
C08309=1057.525,391.553,-117.384,174.534,38.669,157.394
C08310=1057.517,391.307,-117.343,174.529,38.662,157.392
C08311=1057.509,391.060,-117.301,174.522,38.654,157.390
C08312=1057.501,390.814,-117.259,174.516,38.647,157.388
C08313=1057.493,390.568,-117.218,174.510,38.640,157.386
C08314=1057.485,390.321,-117.176,174.504,38.633,157.384
C08315=1057.478,390.075,-117.135,174.498,38.626,157.382
C08316=1057.469,389.829,-117.093,174.492,38.619,157.380
C08317=1057.462,389.582,-117.052,174.485,38.612,157.379
C08318=1057.453,389.336,-117.010,174.480,38.606,157.377
C08319=1057.446,389.089,-116.969,174.474,38.599,157.375
C08320=1057.437,388.844,-116.928,174.468,38.592,157.373
C08321=1057.430,388.597,-116.887,174.462,38.585,157.371
C08322=1057.420,388.283,-116.834,174.454,38.576,157.369
C08323=1057.410,387.969,-116.782,174.446,38.567,157.367
C08324=1057.400,387.654,-116.729,174.439,38.558,157.364
C08325=1057.390,387.340,-116.676,174.431,38.550,157.362
C08326=1057.382,387.094,-116.636,174.425,38.543,157.360
C08327=1057.374,386.847,-116.595,174.419,38.537,157.359
C08328=1057.366,386.601,-116.554,174.413,38.530,157.357
C08329=1057.359,386.354,-116.513,174.408,38.523,157.355
C08330=1057.350,386.107,-116.472,174.401,38.516,157.353
C08331=1057.342,385.861,-116.431,174.396,38.509,157.351
C08332=1057.335,385.615,-116.390,174.390,38.503,157.350
C08333=1057.327,385.368,-116.349,174.384,38.496,157.348
C08334=1057.320,385.122,-116.308,174.378,38.489,157.346
C08335=1057.312,384.875,-116.267,174.373,38.483,157.345
C08336=1057.304,384.629,-116.227,174.367,38.476,157.343
C08337=1057.296,384.382,-116.185,174.361,38.469,157.341
C08338=1057.288,384.136,-116.145,174.355,38.463,157.339
C08339=1057.281,383.890,-116.104,174.350,38.456,157.338
C08340=1057.273,383.643,-116.064,174.343,38.449,157.336
C08341=1057.266,383.397,-116.023,174.338,38.443,157.334
C08342=1057.259,383.151,-115.982,174.332,38.437,157.332
C08343=1057.251,382.904,-115.942,174.327,38.430,157.331
C08344=1057.243,382.657,-115.902,174.322,38.424,157.329
C08345=1057.236,382.411,-115.860,174.315,38.417,157.327
C08346=1057.228,382.164,-115.820,174.310,38.410,157.326
C08347=1057.220,381.918,-115.780,174.304,38.404,157.324
C08348=1057.213,381.671,-115.739,174.299,38.397,157.322
C08349=1057.205,381.425,-115.699,174.292,38.391,157.321
C08350=1057.197,381.178,-115.658,174.287,38.384,157.319
C08351=1057.190,380.931,-115.618,174.282,38.378,157.317
C08352=1057.182,380.685,-115.577,174.276,38.371,157.315
C08353=1057.175,380.439,-115.538,174.271,38.365,157.314
C08354=1057.168,380.192,-115.497,174.265,38.359,157.312
C08355=1057.160,379.945,-115.457,174.259,38.352,157.311
C08356=1057.153,379.698,-115.417,174.254,38.346,157.309
C08357=1057.145,379.452,-115.376,174.248,38.340,157.307
C08358=1057.137,379.205,-115.336,174.243,38.334,157.306
C08359=1057.130,378.959,-115.297,174.238,38.328,157.304
C08360=1057.122,378.712,-115.257,174.232,38.321,157.302
C08361=1057.114,378.466,-115.216,174.226,38.315,157.301
C08362=1057.106,378.219,-115.176,174.220,38.309,157.299
C08363=1057.099,377.973,-115.137,174.215,38.303,157.298
C08364=1057.091,377.726,-115.097,174.210,38.296,157.296
C08365=1057.084,377.479,-115.057,174.205,38.290,157.295
C08366=1057.077,377.233,-115.017,174.199,38.284,157.293
C08367=1057.069,376.986,-114.977,174.194,38.278,157.291
C08368=1057.061,376.739,-114.937,174.188,38.271,157.290
C08369=1057.054,376.493,-114.898,174.183,38.265,157.288
C08370=1057.046,376.246,-114.858,174.178,38.259,157.287
C08371=1057.039,375.999,-114.818,174.173,38.253,157.285
C08372=1057.031,375.753,-114.778,174.166,38.247,157.283
C08373=1057.024,375.506,-114.738,174.161,38.241,157.282
C08374=1057.017,375.260,-114.699,174.156,38.235,157.280
C08375=1057.009,375.013,-114.659,174.150,38.229,157.279
C08376=1057.001,374.765,-114.620,174.145,38.223,157.277
C08377=1056.994,374.519,-114.580,174.140,38.217,157.276
C08378=1056.986,374.236,-114.535,174.134,38.210,157.274
C08379=1056.977,373.953,-114.490,174.128,38.203,157.272
C08380=1056.969,373.671,-114.444,174.122,38.196,157.270
C08381=1056.960,373.389,-114.399,174.116,38.189,157.268
C08382=1056.953,373.142,-114.360,174.111,38.183,157.267
C08383=1056.946,372.895,-114.321,174.105,38.177,157.265
C08384=1056.938,372.648,-114.281,174.100,38.171,157.264
C08385=1056.931,372.402,-114.242,174.095,38.165,157.263
C08386=1056.923,372.155,-114.202,174.090,38.159,157.261
C08387=1056.917,371.908,-114.163,174.085,38.153,157.259
C08388=1056.909,371.661,-114.123,174.079,38.147,157.258
C08389=1056.901,371.414,-114.085,174.074,38.141,157.256
C08390=1056.894,371.168,-114.046,174.069,38.136,157.255
C08391=1056.887,370.921,-114.006,174.064,38.130,157.254
C08392=1056.879,370.674,-113.968,174.059,38.124,157.252
C08393=1056.871,370.427,-113.928,174.053,38.119,157.251
C08394=1056.864,370.181,-113.890,174.048,38.113,157.249
C08395=1056.856,369.933,-113.851,174.044,38.107,157.248
C08396=1056.850,369.686,-113.812,174.039,38.101,157.246
C08397=1056.842,369.441,-113.773,174.034,38.095,157.245
C08398=1056.834,369.193,-113.734,174.028,38.090,157.243
C08399=1056.828,368.946,-113.695,174.023,38.084,157.242
C08400=1056.820,368.700,-113.656,174.018,38.078,157.240
C08401=1056.813,368.452,-113.617,174.013,38.072,157.239
C08402=1056.805,368.206,-113.579,174.008,38.067,157.237
C08403=1056.798,367.959,-113.539,174.003,38.061,157.236
C08404=1056.791,367.713,-113.501,173.997,38.055,157.235
C08405=1056.783,367.465,-113.462,173.993,38.050,157.233
C08406=1056.776,367.219,-113.423,173.988,38.044,157.232
C08407=1056.769,366.972,-113.385,173.983,38.038,157.230
C08408=1056.762,366.725,-113.346,173.978,38.033,157.229
C08409=1056.754,366.478,-113.307,173.973,38.027,157.227
C08410=1056.747,366.231,-113.269,173.968,38.021,157.226
C08411=1056.740,365.984,-113.230,173.963,38.016,157.225
C08412=1056.733,365.737,-113.192,173.958,38.010,157.223
C08413=1056.726,365.490,-113.153,173.953,38.004,157.222
C08414=1056.718,365.243,-113.115,173.948,37.999,157.220
C08415=1056.711,364.996,-113.076,173.943,37.994,157.219
C08416=1056.704,364.750,-113.037,173.939,37.988,157.218
C08417=1056.697,364.503,-112.999,173.934,37.983,157.216
C08418=1056.690,364.256,-112.961,173.929,37.976,157.215
C08419=1056.683,364.009,-112.923,173.923,37.971,157.213
C08420=1056.676,363.762,-112.884,173.918,37.966,157.212
C08421=1056.669,363.515,-112.846,173.914,37.960,157.211
C08422=1056.662,363.268,-112.807,173.909,37.955,157.209
C08423=1056.654,363.021,-112.769,173.904,37.949,157.208
C08424=1056.646,362.774,-112.731,173.899,37.944,157.207
C08425=1056.640,362.527,-112.692,173.895,37.939,157.205
C08426=1056.632,362.280,-112.655,173.890,37.933,157.204
C08427=1056.625,362.033,-112.617,173.885,37.928,157.203
C08428=1056.617,361.786,-112.579,173.880,37.922,157.201
C08429=1056.611,361.540,-112.540,173.876,37.917,157.200
C08430=1056.603,361.292,-112.503,173.871,37.911,157.198
C08431=1056.596,361.046,-112.465,173.866,37.906,157.197
C08432=1056.589,360.798,-112.426,173.861,37.901,157.196
C08433=1056.582,360.551,-112.389,173.857,37.895,157.194
C08434=1056.574,360.287,-112.348,173.851,37.890,157.193
C08435=1056.566,360.024,-112.308,173.846,37.884,157.192
C08436=1056.558,359.759,-112.267,173.841,37.878,157.190
C08437=1056.551,359.495,-112.226,173.836,37.873,157.189
C08438=1056.544,359.248,-112.189,173.831,37.867,157.187
C08439=1056.537,359.000,-112.151,173.827,37.862,157.186
C08440=1056.530,358.753,-112.113,173.822,37.857,157.185
C08441=1056.522,358.507,-112.075,173.817,37.851,157.184
C08442=1056.515,358.260,-112.038,173.813,37.846,157.182
C08443=1056.508,358.013,-112.000,173.808,37.841,157.181
C08444=1056.502,357.766,-111.962,173.803,37.836,157.180
C08445=1056.495,357.519,-111.925,173.799,37.830,157.178
C08446=1056.488,357.272,-111.887,173.794,37.825,157.177
C08447=1056.480,357.024,-111.850,173.789,37.820,157.176
C08448=1056.473,356.777,-111.812,173.785,37.815,157.175
C08449=1056.466,356.530,-111.775,173.780,37.810,157.173
C08450=1056.459,356.283,-111.737,173.775,37.804,157.172
C08451=1056.451,356.036,-111.700,173.771,37.799,157.171
C08452=1056.445,355.789,-111.662,173.766,37.794,157.169
C08453=1056.437,355.542,-111.625,173.761,37.789,157.168
C08454=1056.430,355.295,-111.587,173.757,37.784,157.167
C08455=1056.423,355.048,-111.550,173.752,37.779,157.166
C08456=1056.416,354.800,-111.513,173.748,37.774,157.164
C08457=1056.409,354.554,-111.476,173.743,37.768,157.163
C08458=1056.402,354.307,-111.438,173.738,37.763,157.162
C08459=1056.395,354.060,-111.401,173.734,37.758,157.161
C08460=1056.388,353.812,-111.363,173.729,37.754,157.159
C08461=1056.381,353.565,-111.326,173.725,37.749,157.158
C08462=1056.374,353.318,-111.289,173.721,37.744,157.157
C08463=1056.367,353.071,-111.252,173.716,37.738,157.156
C08464=1056.360,352.823,-111.215,173.712,37.733,157.154
C08465=1056.353,352.577,-111.178,173.708,37.728,157.153
C08466=1056.346,352.330,-111.140,173.703,37.723,157.152
C08467=1056.339,352.082,-111.103,173.698,37.718,157.151
C08468=1056.332,351.836,-111.066,173.694,37.713,157.150
C08469=1056.325,351.588,-111.029,173.689,37.708,157.148
C08470=1056.318,351.341,-110.992,173.685,37.703,157.147
C08471=1056.311,351.094,-110.956,173.680,37.698,157.146
C08472=1056.304,350.847,-110.919,173.676,37.693,157.145
C08473=1056.297,350.599,-110.882,173.671,37.688,157.143
C08474=1056.290,350.353,-110.845,173.667,37.683,157.142
C08475=1056.283,350.105,-110.808,173.662,37.678,157.141
C08476=1056.275,349.858,-110.771,173.659,37.674,157.140
C08477=1056.269,349.611,-110.734,173.654,37.669,157.139
C08478=1056.262,349.363,-110.698,173.650,37.664,157.137
C08479=1056.254,349.116,-110.661,173.645,37.659,157.136
C08480=1056.248,348.869,-110.624,173.641,37.654,157.135
C08481=1056.241,348.622,-110.587,173.636,37.649,157.134
C08482=1056.235,348.375,-110.551,173.632,37.644,157.133
C08483=1056.227,348.128,-110.514,173.627,37.639,157.132
C08484=1056.220,347.881,-110.478,173.623,37.634,157.130
C08485=1056.213,347.633,-110.441,173.618,37.630,157.129
C08486=1056.206,347.385,-110.404,173.615,37.625,157.128
C08487=1056.199,347.138,-110.368,173.611,37.620,157.127
C08488=1056.192,346.891,-110.331,173.606,37.615,157.126
C08489=1056.186,346.644,-110.294,173.602,37.610,157.125
C08490=1056.178,346.385,-110.256,173.597,37.605,157.123
C08491=1056.171,346.125,-110.218,173.592,37.600,157.122
C08492=1056.163,345.866,-110.180,173.588,37.595,157.121
C08493=1056.157,345.607,-110.141,173.583,37.590,157.120
C08494=1056.150,345.360,-110.106,173.579,37.585,157.118
C08495=1056.143,345.112,-110.069,173.575,37.581,157.117
C08496=1056.136,344.865,-110.033,173.571,37.576,157.116
C08497=1056.129,344.618,-109.997,173.567,37.571,157.115
C08498=1056.122,344.370,-109.960,173.562,37.566,157.114
C08499=1056.115,344.124,-109.924,173.558,37.561,157.113
C08500=1056.108,343.876,-109.887,173.554,37.557,157.112
C08501=1056.101,343.629,-109.851,173.549,37.552,157.110
C08502=1056.095,343.382,-109.815,173.546,37.547,157.109
C08503=1056.088,343.134,-109.779,173.541,37.543,157.108
C08504=1056.081,342.887,-109.743,173.537,37.538,157.107
C08505=1056.073,342.640,-109.707,173.533,37.533,157.106
C08506=1056.067,342.393,-109.670,173.528,37.529,157.105
C08507=1056.060,342.145,-109.635,173.524,37.524,157.104
C08508=1056.053,341.897,-109.598,173.521,37.519,157.103
C08509=1056.046,341.651,-109.562,173.516,37.515,157.102
C08510=1056.039,341.403,-109.527,173.512,37.510,157.100
C08511=1056.033,341.156,-109.490,173.508,37.505,157.099
C08512=1056.026,340.909,-109.455,173.503,37.501,157.098
C08513=1056.018,340.661,-109.419,173.500,37.497,157.097
C08514=1056.012,340.414,-109.383,173.495,37.491,157.096
C08515=1056.005,340.166,-109.347,173.491,37.487,157.095
C08516=1055.998,339.920,-109.312,173.487,37.483,157.094
C08517=1055.991,339.671,-109.276,173.483,37.478,157.093
C08518=1055.984,339.424,-109.240,173.479,37.474,157.092
C08519=1055.978,339.177,-109.204,173.475,37.469,157.090
C08520=1055.971,338.929,-109.168,173.471,37.464,157.089
C08521=1055.964,338.682,-109.133,173.466,37.460,157.088
C08522=1055.957,338.435,-109.096,173.462,37.455,157.087
C08523=1055.951,338.188,-109.061,173.459,37.451,157.086
C08524=1055.944,337.940,-109.026,173.454,37.446,157.085
C08525=1055.936,337.693,-108.990,173.450,37.442,157.084
C08526=1055.930,337.445,-108.954,173.446,37.437,157.083
C08527=1055.923,337.198,-108.918,173.443,37.433,157.082
C08528=1055.916,336.951,-108.883,173.438,37.428,157.081
C08529=1055.910,336.703,-108.847,173.434,37.423,157.080
C08530=1055.903,336.455,-108.812,173.430,37.419,157.079
C08531=1055.896,336.208,-108.776,173.426,37.414,157.077
C08532=1055.889,335.961,-108.741,173.422,37.410,157.076
C08533=1055.882,335.714,-108.706,173.418,37.406,157.075
C08534=1055.876,335.466,-108.670,173.414,37.401,157.074
C08535=1055.869,335.219,-108.635,173.410,37.397,157.073
C08536=1055.862,334.971,-108.599,173.406,37.392,157.072
C08537=1055.855,334.724,-108.563,173.402,37.388,157.071
C08538=1055.848,334.477,-108.528,173.398,37.383,157.070
C08539=1055.842,334.229,-108.493,173.394,37.379,157.069
C08540=1055.835,333.982,-108.458,173.390,37.375,157.068
C08541=1055.828,333.734,-108.423,173.386,37.370,157.067
C08542=1055.821,333.487,-108.388,173.382,37.366,157.066
C08543=1055.815,333.240,-108.353,173.378,37.361,157.065
C08544=1055.808,332.992,-108.317,173.375,37.357,157.064
C08545=1055.801,332.745,-108.282,173.370,37.352,157.063
C08546=1055.794,332.481,-108.245,173.366,37.348,157.062
C08547=1055.787,332.217,-108.207,173.362,37.343,157.061
C08548=1055.780,331.954,-108.170,173.358,37.339,157.060
C08549=1055.772,331.690,-108.133,173.354,37.334,157.058
C08550=1055.766,331.443,-108.097,173.350,37.330,157.057
C08551=1055.759,331.195,-108.062,173.346,37.325,157.056
C08552=1055.752,330.948,-108.027,173.342,37.321,157.055
C08553=1055.745,330.701,-107.992,173.338,37.316,157.054
C08554=1055.738,330.453,-107.957,173.334,37.312,157.053
C08555=1055.733,330.206,-107.923,173.330,37.308,157.052
C08556=1055.725,329.958,-107.887,173.327,37.303,157.051
C08557=1055.718,329.711,-107.853,173.323,37.299,157.050
C08558=1055.711,329.463,-107.818,173.318,37.295,157.049
C08559=1055.704,329.215,-107.783,173.315,37.291,157.048
C08560=1055.697,328.968,-107.749,173.311,37.287,157.047
C08561=1055.691,328.720,-107.714,173.307,37.282,157.046
C08562=1055.684,328.473,-107.679,173.304,37.278,157.045
C08563=1055.677,328.225,-107.645,173.300,37.274,157.044
C08564=1055.670,327.978,-107.610,173.296,37.270,157.043
C08565=1055.663,327.730,-107.576,173.291,37.265,157.042
C08566=1055.656,327.483,-107.541,173.288,37.262,157.041
C08567=1055.650,327.236,-107.507,173.284,37.257,157.040
C08568=1055.643,326.988,-107.472,173.280,37.253,157.039
C08569=1055.636,326.741,-107.438,173.277,37.249,157.039
C08570=1055.629,326.493,-107.403,173.273,37.245,157.037
C08571=1055.623,326.245,-107.369,173.269,37.241,157.037
C08572=1055.615,325.998,-107.334,173.266,37.236,157.035
C08573=1055.609,325.750,-107.300,173.262,37.232,157.035
C08574=1055.602,325.503,-107.265,173.257,37.228,157.034
C08575=1055.595,325.255,-107.231,173.254,37.224,157.033
C08576=1055.589,325.008,-107.197,173.250,37.220,157.032
C08577=1055.581,324.761,-107.162,173.246,37.216,157.031
C08578=1055.575,324.513,-107.128,173.243,37.211,157.030
C08579=1055.569,324.265,-107.093,173.239,37.207,157.029
C08580=1055.561,324.017,-107.059,173.235,37.203,157.028
C08581=1055.555,323.770,-107.024,173.232,37.199,157.027
C08582=1055.548,323.523,-106.991,173.228,37.195,157.026
C08583=1055.541,323.275,-106.956,173.224,37.191,157.025
C08584=1055.535,323.027,-106.922,173.221,37.187,157.024
C08585=1055.528,322.780,-106.887,173.217,37.182,157.023
C08586=1055.522,322.533,-106.853,173.213,37.178,157.022
C08587=1055.514,322.285,-106.820,173.210,37.174,157.021
C08588=1055.508,322.037,-106.785,173.206,37.170,157.020
C08589=1055.501,321.789,-106.751,173.202,37.166,157.019
C08590=1055.495,321.542,-106.717,173.199,37.162,157.018
C08591=1055.488,321.295,-106.682,173.195,37.158,157.017
C08592=1055.481,321.047,-106.648,173.191,37.154,157.016
C08593=1055.475,320.800,-106.614,173.188,37.149,157.015
C08594=1055.468,320.552,-106.580,173.184,37.145,157.014
C08595=1055.461,320.304,-106.546,173.180,37.141,157.013
C08596=1055.455,320.057,-106.513,173.177,37.137,157.013
C08597=1055.448,319.809,-106.478,173.173,37.133,157.012
C08598=1055.441,319.561,-106.444,173.169,37.129,157.011
C08599=1055.435,319.314,-106.410,173.166,37.125,157.010
C08600=1055.429,319.066,-106.376,173.162,37.121,157.009
C08601=1055.422,318.819,-106.342,173.158,37.117,157.008
C08602=1055.415,318.550,-106.305,173.155,37.112,157.007
C08603=1055.408,318.280,-106.269,173.150,37.108,157.006
C08604=1055.401,318.012,-106.232,173.146,37.104,157.005
C08605=1055.394,317.743,-106.195,173.143,37.099,157.004
C08606=1055.388,317.496,-106.161,173.139,37.095,157.003
C08607=1055.380,317.248,-106.127,173.135,37.091,157.002
C08608=1055.375,317.001,-106.093,173.132,37.087,157.001
C08609=1055.368,316.753,-106.060,173.128,37.083,157.000
C08610=1055.362,316.505,-106.026,173.125,37.079,156.999
C08611=1055.355,316.258,-105.992,173.121,37.075,156.998
C08612=1055.349,316.010,-105.958,173.117,37.071,156.997
C08613=1055.342,315.763,-105.924,173.114,37.067,156.996
C08614=1055.336,315.515,-105.891,173.111,37.063,156.995
C08615=1055.329,315.267,-105.857,173.107,37.059,156.994
C08616=1055.323,315.020,-105.823,173.104,37.055,156.994
C08617=1055.316,314.772,-105.790,173.100,37.051,156.993
C08618=1055.310,314.524,-105.756,173.097,37.047,156.992
C08619=1055.303,314.277,-105.722,173.093,37.043,156.991
C08620=1055.297,314.029,-105.689,173.089,37.038,156.990
C08621=1055.291,313.782,-105.655,173.086,37.034,156.989
C08622=1055.284,313.534,-105.622,173.082,37.030,156.988
C08623=1055.278,313.286,-105.588,173.079,37.026,156.987
C08624=1055.271,313.038,-105.554,173.076,37.023,156.986
C08625=1055.265,312.791,-105.522,173.072,37.019,156.985
C08626=1055.258,312.543,-105.489,173.069,37.015,156.984
C08627=1055.251,312.296,-105.455,173.065,37.011,156.984
C08628=1055.244,312.047,-105.422,173.062,37.007,156.983
C08629=1055.238,311.800,-105.389,173.058,37.003,156.982
C08630=1055.231,311.552,-105.355,173.054,36.999,156.981
C08631=1055.224,311.305,-105.323,173.051,36.995,156.980
C08632=1055.216,311.057,-105.289,173.047,36.992,156.979
C08633=1055.210,310.810,-105.257,173.045,36.988,156.978
C08634=1055.204,310.562,-105.224,173.041,36.984,156.977
C08635=1055.197,310.314,-105.190,173.037,36.981,156.977
C08636=1055.190,310.067,-105.157,173.034,36.977,156.976
C08637=1055.184,309.818,-105.124,173.030,36.973,156.975
C08638=1055.177,309.571,-105.091,173.027,36.968,156.974
C08639=1055.170,309.323,-105.058,173.023,36.965,156.973
C08640=1055.164,309.075,-105.025,173.020,36.961,156.972
C08641=1055.157,308.828,-104.992,173.017,36.957,156.971
C08642=1055.151,308.580,-104.959,173.013,36.954,156.970
C08643=1055.144,308.333,-104.926,173.010,36.950,156.970
C08644=1055.137,308.085,-104.894,173.006,36.946,156.969
C08645=1055.130,307.837,-104.860,173.003,36.942,156.968
C08646=1055.124,307.589,-104.828,172.999,36.938,156.967
C08647=1055.117,307.342,-104.795,172.997,36.934,156.966
C08648=1055.111,307.094,-104.762,172.993,36.931,156.965
C08649=1055.104,306.846,-104.729,172.989,36.927,156.964
C08650=1055.098,306.598,-104.696,172.986,36.923,156.963
C08651=1055.091,306.351,-104.663,172.982,36.919,156.963
C08652=1055.084,306.103,-104.630,172.979,36.915,156.962
C08653=1055.077,305.856,-104.598,172.976,36.912,156.961
C08654=1055.071,305.608,-104.565,172.973,36.908,156.960
C08655=1055.065,305.361,-104.532,172.969,36.904,156.959
C08656=1055.059,305.113,-104.499,172.966,36.900,156.958
C08657=1055.052,304.865,-104.466,172.962,36.896,156.957
C08658=1055.045,304.600,-104.432,172.958,36.892,156.957
C08659=1055.038,304.336,-104.397,172.956,36.888,156.956
C08660=1055.030,304.071,-104.362,172.952,36.884,156.955
C08661=1055.024,303.807,-104.327,172.949,36.880,156.954
C08662=1055.017,303.559,-104.295,172.945,36.876,156.953
C08663=1055.011,303.311,-104.262,172.941,36.873,156.952
C08664=1055.005,303.063,-104.230,172.938,36.869,156.951
C08665=1054.999,302.816,-104.197,172.935,36.865,156.951
C08666=1054.992,302.567,-104.164,172.932,36.861,156.950
C08667=1054.985,302.320,-104.132,172.928,36.857,156.949
C08668=1054.978,302.072,-104.099,172.925,36.854,156.948
C08669=1054.972,301.825,-104.066,172.922,36.850,156.947
C08670=1054.966,301.577,-104.034,172.919,36.846,156.946
C08671=1054.960,301.329,-104.002,172.915,36.842,156.945
C08672=1054.954,301.081,-103.969,172.912,36.839,156.945
C08673=1054.947,300.834,-103.937,172.909,36.835,156.944
C08674=1054.941,300.586,-103.905,172.905,36.831,156.943
C08675=1054.934,300.338,-103.872,172.902,36.827,156.942
C08676=1054.927,300.090,-103.839,172.899,36.823,156.941
C08677=1054.921,299.842,-103.807,172.896,36.820,156.940
C08678=1054.914,299.594,-103.775,172.892,36.816,156.939
C08679=1054.908,299.347,-103.742,172.890,36.812,156.939
C08680=1054.902,299.099,-103.710,172.886,36.808,156.938
C08681=1054.896,298.851,-103.677,172.883,36.805,156.937
C08682=1054.890,298.603,-103.645,172.880,36.801,156.936
C08683=1054.883,298.356,-103.613,172.877,36.797,156.935
C08684=1054.876,298.108,-103.580,172.873,36.793,156.934
C08685=1054.870,297.860,-103.548,172.870,36.790,156.934
C08686=1054.864,297.612,-103.515,172.867,36.786,156.933
C08687=1054.857,297.364,-103.484,172.863,36.782,156.932
C08688=1054.852,297.117,-103.452,172.861,36.778,156.931
C08689=1054.846,296.869,-103.420,172.857,36.774,156.930
C08690=1054.840,296.622,-103.387,172.854,36.771,156.929
C08691=1054.833,296.374,-103.355,172.851,36.767,156.929
C08692=1054.827,296.125,-103.323,172.848,36.763,156.928
C08693=1054.820,295.878,-103.291,172.844,36.760,156.927
C08694=1054.814,295.630,-103.259,172.842,36.756,156.926
C08695=1054.807,295.382,-103.228,172.838,36.752,156.925
C08696=1054.801,295.134,-103.195,172.835,36.749,156.924
C08697=1054.794,294.887,-103.164,172.832,36.745,156.924
C08698=1054.788,294.638,-103.132,172.829,36.741,156.923
C08699=1054.781,294.391,-103.099,172.825,36.738,156.922
C08700=1054.774,294.143,-103.068,172.823,36.734,156.921
C08701=1054.768,293.895,-103.036,172.819,36.730,156.920
C08702=1054.762,293.647,-103.005,172.816,36.727,156.920
C08703=1054.756,293.399,-102.973,172.813,36.723,156.919
C08704=1054.749,293.152,-102.940,172.810,36.719,156.918
C08705=1054.742,292.904,-102.909,172.807,36.716,156.917
C08706=1054.736,292.655,-102.877,172.804,36.712,156.916
C08707=1054.729,292.408,-102.846,172.800,36.709,156.916
C08708=1054.722,292.160,-102.814,172.798,36.705,156.915
C08709=1054.716,291.911,-102.782,172.794,36.701,156.914
C08710=1054.710,291.664,-102.751,172.792,36.698,156.913
C08711=1054.703,291.417,-102.719,172.788,36.694,156.912
C08712=1054.697,291.169,-102.687,172.785,36.690,156.912
C08713=1054.691,290.921,-102.655,172.782,36.687,156.911
C08714=1054.684,290.671,-102.624,172.779,36.683,156.910
C08715=1054.678,290.423,-102.592,172.776,36.679,156.909
C08716=1054.671,290.174,-102.561,172.773,36.676,156.908
C08717=1054.665,289.926,-102.529,172.769,36.672,156.908
C08718=1054.659,289.678,-102.497,172.767,36.669,156.907
C08719=1054.652,289.430,-102.466,172.763,36.665,156.906
C08720=1054.645,289.182,-102.434,172.761,36.661,156.905
C08721=1054.639,288.934,-102.402,172.757,36.658,156.904
C08722=1054.632,288.686,-102.371,172.754,36.654,156.904
C08723=1054.627,288.438,-102.340,172.751,36.651,156.903
C08724=1054.620,288.190,-102.309,172.748,36.647,156.902
C08725=1054.613,287.942,-102.278,172.745,36.643,156.901
C08726=1054.607,287.694,-102.246,172.742,36.640,156.900
C08727=1054.600,287.446,-102.214,172.739,36.636,156.900
C08728=1054.594,287.198,-102.183,172.736,36.633,156.899
C08729=1054.588,286.950,-102.152,172.733,36.629,156.898
C08730=1054.581,286.702,-102.121,172.730,36.626,156.897
C08731=1054.574,286.455,-102.089,172.726,36.622,156.897
C08732=1054.568,286.207,-102.058,172.724,36.619,156.896
C08733=1054.561,285.958,-102.027,172.720,36.615,156.895
C08734=1054.555,285.711,-101.996,172.718,36.611,156.894
C08735=1054.548,285.463,-101.965,172.714,36.608,156.893
C08736=1054.542,285.214,-101.934,172.712,36.604,156.893
C08737=1054.535,284.967,-101.903,172.709,36.601,156.892
C08738=1054.529,284.719,-101.872,172.706,36.597,156.891
C08739=1054.523,284.471,-101.841,172.703,36.594,156.890
C08740=1054.516,284.223,-101.809,172.700,36.590,156.890
C08741=1054.509,283.975,-101.778,172.697,36.587,156.889
C08742=1054.503,283.727,-101.748,172.694,36.583,156.888
C08743=1054.497,283.479,-101.716,172.691,36.579,156.887
C08744=1054.490,283.231,-101.686,172.688,36.576,156.886
C08745=1054.484,282.984,-101.654,172.685,36.572,156.886
C08746=1054.477,282.736,-101.623,172.682,36.569,156.885
C08747=1054.471,282.487,-101.592,172.679,36.565,156.884
C08748=1054.465,282.240,-101.561,172.676,36.562,156.883
C08749=1054.459,281.991,-101.531,172.673,36.558,156.883
C08750=1054.452,281.744,-101.499,172.670,36.555,156.882
C08751=1054.446,281.496,-101.469,172.667,36.551,156.881
C08752=1054.439,281.248,-101.437,172.665,36.548,156.880
C08753=1054.433,280.999,-101.407,172.661,36.544,156.879
C08754=1054.427,280.751,-101.376,172.659,36.540,156.879
C08755=1054.420,280.504,-101.345,172.656,36.537,156.878
C08756=1054.414,280.256,-101.314,172.653,36.533,156.877
C08757=1054.408,280.008,-101.283,172.650,36.530,156.876
C08758=1054.401,279.759,-101.252,172.647,36.526,156.876
C08759=1054.396,279.511,-101.222,172.644,36.523,156.875
C08760=1054.389,279.264,-101.191,172.641,36.519,156.874
C08761=1054.382,279.015,-101.160,172.638,36.516,156.873
C08762=1054.377,278.767,-101.129,172.635,36.512,156.873
C08763=1054.369,278.520,-101.099,172.632,36.509,156.872
C08764=1054.363,278.272,-101.068,172.630,36.505,156.871
C08765=1054.357,278.023,-101.038,172.627,36.501,156.870
C08766=1054.350,277.780,-101.007,172.624,36.498,156.869
C08767=1054.345,277.538,-100.978,172.621,36.494,156.869
C08768=1054.337,277.295,-100.948,172.618,36.492,156.868
C08769=1054.332,277.052,-100.918,172.616,36.488,156.867
C08770=1054.325,276.809,-100.888,172.612,36.485,156.867
C08771=1054.319,276.567,-100.858,172.610,36.481,156.866
C08772=1054.313,276.324,-100.828,172.607,36.478,156.865
C08773=1054.307,276.081,-100.798,172.604,36.474,156.864
C08774=1054.300,275.833,-100.768,172.602,36.470,156.864
C08775=1054.294,275.585,-100.738,172.598,36.467,156.863
C08776=1054.288,275.337,-100.707,172.596,36.463,156.862
C08777=1054.281,275.089,-100.677,172.593,36.460,156.861
C08778=1054.275,274.841,-100.646,172.590,36.456,156.860
C08779=1054.268,274.592,-100.616,172.587,36.453,156.860
C08780=1054.263,274.344,-100.585,172.584,36.450,156.859
C08781=1054.255,274.096,-100.555,172.582,36.446,156.858
C08782=1054.250,273.848,-100.525,172.579,36.443,156.858
C08783=1054.243,273.600,-100.494,172.576,36.439,156.857
C08784=1054.237,273.352,-100.464,172.573,36.436,156.856
C08785=1054.231,273.104,-100.434,172.571,36.432,156.855
C08786=1054.224,272.856,-100.404,172.567,36.429,156.855
C08787=1054.218,272.608,-100.373,172.565,36.425,156.854
C08788=1054.211,272.360,-100.343,172.561,36.422,156.853
C08789=1054.205,272.112,-100.313,172.559,36.418,156.852
C08790=1054.198,271.864,-100.282,172.557,36.415,156.852
C08791=1054.192,271.616,-100.253,172.553,36.411,156.851
C08792=1054.185,271.368,-100.222,172.551,36.408,156.850
C08793=1054.179,271.120,-100.193,172.548,36.404,156.849
C08794=1054.173,270.871,-100.162,172.545,36.401,156.849
C08795=1054.166,270.623,-100.132,172.542,36.398,156.848
C08796=1054.160,270.375,-100.102,172.540,36.394,156.847
C08797=1054.153,270.127,-100.072,172.537,36.391,156.846
C08798=1054.148,269.879,-100.042,172.534,36.387,156.846
C08799=1054.141,269.631,-100.012,172.532,36.384,156.845
C08800=1054.135,269.383,-99.982,172.528,36.380,156.844
C08801=1054.128,269.135,-99.952,172.526,36.377,156.843
C08802=1054.122,268.886,-99.922,172.523,36.373,156.843
C08803=1054.116,268.639,-99.892,172.520,36.370,156.842
C08804=1054.109,268.390,-99.861,172.518,36.367,156.841
C08805=1054.103,268.142,-99.832,172.515,36.363,156.840
C08806=1054.096,267.894,-99.802,172.512,36.360,156.840
C08807=1054.090,267.646,-99.772,172.509,36.356,156.839
C08808=1054.084,267.398,-99.743,172.507,36.353,156.838
C08809=1054.077,267.149,-99.712,172.504,36.349,156.837
C08810=1054.071,266.901,-99.683,172.501,36.346,156.837
C08811=1054.064,266.654,-99.653,172.499,36.343,156.836
C08812=1054.058,266.405,-99.623,172.496,36.339,156.835
C08813=1054.052,266.157,-99.594,172.493,36.336,156.835
C08814=1054.045,265.909,-99.564,172.490,36.332,156.834
C08815=1054.039,265.660,-99.534,172.488,36.328,156.833
C08816=1054.033,265.413,-99.504,172.485,36.325,156.832
C08817=1054.026,265.165,-99.475,172.482,36.322,156.832
C08818=1054.020,264.916,-99.444,172.480,36.318,156.831
C08819=1054.014,264.668,-99.415,172.477,36.315,156.830
C08820=1054.007,264.421,-99.386,172.474,36.311,156.829
C08821=1054.001,264.172,-99.356,172.471,36.308,156.829
C08822=1053.995,263.931,-99.328,172.469,36.304,156.828
C08823=1053.989,263.690,-99.298,172.467,36.301,156.827
C08824=1053.983,263.450,-99.270,172.464,36.298,156.827
C08825=1053.976,263.209,-99.241,172.461,36.294,156.826
C08826=1053.970,262.968,-99.212,172.458,36.291,156.825
C08827=1053.964,262.727,-99.184,172.456,36.288,156.824
C08828=1053.957,262.486,-99.155,172.454,36.285,156.824
C08829=1053.951,262.245,-99.126,172.451,36.281,156.823
C08830=1053.945,261.997,-99.097,172.448,36.278,156.822
C08831=1053.939,261.749,-99.068,172.445,36.275,156.822
C08832=1053.932,261.500,-99.038,172.443,36.271,156.821
C08833=1053.925,261.253,-99.009,172.441,36.268,156.820
C08834=1053.919,261.005,-98.980,172.437,36.265,156.820
C08835=1053.912,260.756,-98.950,172.435,36.261,156.819
C08836=1053.906,260.508,-98.921,172.432,36.258,156.818
C08837=1053.899,260.260,-98.893,172.430,36.254,156.817
C08838=1053.892,260.012,-98.863,172.427,36.251,156.817
C08839=1053.886,259.764,-98.834,172.424,36.248,156.816
C08840=1053.879,259.515,-98.805,172.422,36.244,156.815
C08841=1053.873,259.267,-98.775,172.420,36.241,156.815
C08842=1053.867,259.019,-98.746,172.417,36.238,156.814
C08843=1053.860,258.770,-98.717,172.414,36.234,156.813
C08844=1053.854,258.522,-98.688,172.411,36.231,156.812
C08845=1053.847,258.274,-98.659,172.409,36.228,156.812
C08846=1053.841,258.027,-98.629,172.406,36.224,156.811
C08847=1053.834,257.778,-98.600,172.403,36.220,156.810
C08848=1053.828,257.530,-98.571,172.401,36.218,156.810
C08849=1053.822,257.281,-98.542,172.398,36.214,156.809
C08850=1053.815,257.033,-98.513,172.396,36.210,156.808
C08851=1053.809,256.785,-98.484,172.394,36.207,156.807
C08852=1053.803,256.537,-98.455,172.391,36.204,156.807
C08853=1053.796,256.288,-98.425,172.388,36.200,156.806
C08854=1053.790,256.040,-98.396,172.385,36.197,156.805
C08855=1053.783,255.792,-98.368,172.383,36.193,156.804
C08856=1053.776,255.544,-98.339,172.381,36.190,156.804
C08857=1053.770,255.296,-98.310,172.378,36.187,156.803
C08858=1053.764,255.047,-98.281,172.375,36.183,156.802
C08859=1053.758,254.799,-98.252,172.372,36.180,156.802
C08860=1053.751,254.550,-98.223,172.370,36.177,156.801
C08861=1053.745,254.302,-98.194,172.368,36.173,156.800
C08862=1053.739,254.054,-98.165,172.365,36.170,156.799
C08863=1053.732,253.806,-98.136,172.363,36.166,156.799
C08864=1053.726,253.558,-98.107,172.360,36.163,156.798
C08865=1053.720,253.310,-98.078,172.357,36.160,156.797
C08866=1053.713,253.061,-98.050,172.355,36.156,156.797
C08867=1053.707,252.813,-98.021,172.352,36.152,156.796
C08868=1053.701,252.565,-97.992,172.350,36.149,156.795
C08869=1053.694,252.317,-97.963,172.348,36.146,156.794
C08870=1053.688,252.069,-97.934,172.345,36.142,156.794
C08871=1053.682,251.820,-97.905,172.343,36.139,156.793
C08872=1053.676,251.572,-97.876,172.340,36.135,156.792
C08873=1053.669,251.323,-97.847,172.337,36.132,156.791
C08874=1053.663,251.075,-97.818,172.335,36.129,156.791
C08875=1053.656,250.826,-97.790,172.332,36.125,156.790
C08876=1053.650,250.578,-97.761,172.330,36.122,156.789
C08877=1053.644,250.330,-97.732,172.327,36.118,156.789
C08878=1053.638,250.088,-97.704,172.325,36.115,156.788
C08879=1053.632,249.847,-97.677,172.323,36.112,156.787
C08880=1053.626,249.606,-97.648,172.320,36.108,156.787
C08881=1053.620,249.364,-97.620,172.318,36.105,156.786
C08882=1053.614,249.122,-97.593,172.316,36.101,156.785
C08883=1053.608,248.880,-97.565,172.313,36.098,156.784
C08884=1053.601,248.638,-97.537,172.311,36.094,156.784
C08885=1053.596,248.396,-97.509,172.308,36.091,156.783
C08886=1053.590,248.148,-97.480,172.306,36.088,156.782
C08887=1053.583,247.900,-97.452,172.304,36.084,156.782
C08888=1053.577,247.652,-97.423,172.301,36.081,156.781
C08889=1053.570,247.403,-97.394,172.299,36.077,156.780
C08890=1053.564,247.155,-97.366,172.296,36.074,156.779
C08891=1053.559,246.907,-97.337,172.294,36.071,156.779
C08892=1053.553,246.658,-97.309,172.291,36.067,156.778
C08893=1053.546,246.411,-97.280,172.288,36.063,156.777
C08894=1053.540,246.162,-97.252,172.286,36.060,156.776
C08895=1053.534,245.914,-97.223,172.284,36.056,156.776
C08896=1053.528,245.665,-97.195,172.281,36.053,156.775
C08897=1053.521,245.417,-97.166,172.279,36.050,156.774
C08898=1053.515,245.168,-97.138,172.276,36.046,156.774
C08899=1053.508,244.920,-97.110,172.274,36.043,156.773
C08900=1053.502,244.672,-97.081,172.272,36.040,156.772
C08901=1053.496,244.423,-97.053,172.269,36.036,156.772
C08902=1053.489,244.175,-97.024,172.267,36.033,156.771
C08903=1053.484,243.927,-96.996,172.265,36.029,156.770
C08904=1053.477,243.679,-96.969,172.262,36.025,156.769
C08905=1053.471,243.431,-96.940,172.260,36.022,156.769
C08906=1053.465,243.182,-96.911,172.257,36.019,156.768
C08907=1053.458,242.933,-96.883,172.255,36.015,156.767
C08908=1053.452,242.685,-96.855,172.253,36.012,156.766
C08909=1053.445,242.437,-96.827,172.250,36.009,156.766
C08910=1053.439,242.188,-96.798,172.248,36.005,156.765
C08911=1053.433,241.940,-96.771,172.246,36.002,156.764
C08912=1053.427,241.692,-96.742,172.243,35.998,156.764
C08913=1053.420,241.444,-96.714,172.241,35.995,156.763
C08914=1053.414,241.195,-96.686,172.238,35.991,156.762
C08915=1053.408,240.947,-96.658,172.236,35.988,156.762
C08916=1053.401,240.698,-96.630,172.234,35.984,156.761
C08917=1053.395,240.449,-96.602,172.231,35.981,156.760
C08918=1053.388,240.202,-96.574,172.229,35.978,156.759
C08919=1053.382,239.954,-96.546,172.227,35.974,156.759
C08920=1053.376,239.705,-96.518,172.224,35.971,156.758
C08921=1053.369,239.457,-96.490,172.222,35.968,156.757
C08922=1053.363,239.208,-96.462,172.220,35.964,156.757
C08923=1053.357,238.959,-96.434,172.217,35.961,156.756
C08924=1053.350,238.711,-96.406,172.215,35.958,156.755
C08925=1053.345,238.463,-96.379,172.212,35.954,156.755
C08926=1053.338,238.215,-96.351,172.210,35.950,156.754
C08927=1053.331,237.966,-96.323,172.208,35.947,156.753
C08928=1053.325,237.718,-96.295,172.205,35.944,156.752
C08929=1053.319,237.469,-96.267,172.203,35.940,156.752
C08930=1053.313,237.221,-96.240,172.201,35.937,156.751
C08931=1053.306,236.973,-96.212,172.198,35.934,156.750
C08932=1053.299,236.724,-96.184,172.196,35.930,156.750
C08933=1053.293,236.476,-96.156,172.194,35.927,156.749
C08934=1053.287,236.231,-96.128,172.191,35.923,156.748
C08935=1053.281,235.986,-96.101,172.189,35.920,156.748
C08936=1053.274,235.741,-96.073,172.188,35.916,156.747
C08937=1053.268,235.498,-96.047,172.185,35.913,156.746
C08938=1053.262,235.253,-96.019,172.183,35.910,156.745
C08939=1053.256,235.008,-95.992,172.181,35.906,156.745
C08940=1053.250,234.763,-95.965,172.178,35.903,156.744
C08941=1053.243,234.518,-95.938,172.176,35.900,156.743
C08942=1053.237,234.270,-95.910,172.173,35.896,156.743
C08943=1053.231,234.021,-95.882,172.171,35.892,156.742
C08944=1053.225,233.773,-95.854,172.169,35.889,156.741
C08945=1053.218,233.525,-95.827,172.166,35.885,156.740
C08946=1053.211,233.276,-95.799,172.164,35.882,156.740
C08947=1053.206,233.028,-95.772,172.163,35.879,156.739
C08948=1053.200,232.779,-95.744,172.160,35.875,156.738
C08949=1053.193,232.531,-95.716,172.158,35.872,156.738
C08950=1053.187,232.283,-95.689,172.156,35.868,156.737
C08951=1053.181,232.034,-95.662,172.153,35.865,156.736
C08952=1053.174,231.785,-95.634,172.151,35.861,156.735
C08953=1053.167,231.537,-95.606,172.149,35.858,156.735
C08954=1053.162,231.289,-95.578,172.146,35.854,156.734
C08955=1053.155,231.040,-95.551,172.144,35.851,156.733
C08956=1053.149,230.792,-95.524,172.142,35.848,156.733
C08957=1053.143,230.544,-95.496,172.140,35.844,156.732
C08958=1053.136,230.295,-95.469,172.138,35.841,156.731
C08959=1053.130,230.047,-95.442,172.135,35.838,156.731
C08960=1053.124,229.798,-95.414,172.133,35.834,156.730
C08961=1053.117,229.549,-95.387,172.131,35.830,156.729
C08962=1053.111,229.302,-95.360,172.128,35.827,156.728
C08963=1053.105,229.053,-95.333,172.126,35.823,156.728
C08964=1053.098,228.804,-95.305,172.124,35.820,156.727
C08965=1053.092,228.556,-95.278,172.122,35.817,156.726
C08966=1053.086,228.307,-95.251,172.120,35.813,156.726
C08967=1053.079,228.059,-95.223,172.118,35.809,156.725
C08968=1053.073,227.811,-95.196,172.115,35.806,156.724
C08969=1053.066,227.562,-95.169,172.113,35.803,156.723
C08970=1053.060,227.313,-95.142,172.111,35.799,156.723
C08971=1053.053,227.066,-95.115,172.108,35.796,156.722
C08972=1053.047,226.817,-95.088,172.107,35.793,156.721
C08973=1053.041,226.568,-95.061,172.105,35.789,156.721
C08974=1053.034,226.320,-95.033,172.102,35.785,156.720
C08975=1053.028,226.071,-95.006,172.100,35.782,156.719
C08976=1053.022,225.823,-94.979,172.098,35.779,156.719
C08977=1053.016,225.574,-94.952,172.095,35.775,156.718
C08978=1053.005,225.180,-94.910,172.092,35.770,156.717
C08979=1052.995,224.785,-94.866,172.088,35.764,156.716
C08980=1052.985,224.390,-94.823,172.086,35.758,156.714
C08981=1052.975,223.995,-94.780,172.082,35.753,156.713
C08982=1052.969,223.747,-94.753,172.080,35.750,156.713
C08983=1052.962,223.498,-94.727,172.077,35.746,156.712
C08984=1052.956,223.250,-94.699,172.075,35.743,156.711
C08985=1052.950,223.001,-94.672,172.073,35.739,156.711
C08986=1052.944,222.753,-94.646,172.071,35.736,156.710
C08987=1052.937,222.504,-94.618,172.069,35.732,156.709
C08988=1052.932,222.256,-94.591,172.067,35.729,156.708
C08989=1052.924,222.007,-94.565,172.064,35.726,156.708
C08990=1052.916,221.657,-94.527,172.062,35.720,156.707
C08991=1052.907,221.306,-94.488,172.058,35.715,156.706
C08992=1052.898,220.954,-94.451,172.056,35.711,156.705
C08993=1052.889,220.604,-94.413,172.053,35.706,156.704
C08994=1052.883,220.356,-94.386,172.050,35.702,156.703
C08995=1052.877,220.107,-94.359,172.049,35.699,156.702
C08996=1052.870,219.858,-94.333,172.046,35.695,156.702
C08997=1052.863,219.610,-94.306,172.044,35.692,156.701
C08998=1052.858,219.362,-94.279,172.042,35.688,156.700
C08999=1052.850,219.113,-94.253,172.041,35.685,156.699
C09000=1052.845,218.865,-94.226,172.038,35.681,156.699
C09001=1052.838,218.616,-94.200,172.036,35.678,156.698
C09002=1052.832,218.367,-94.173,172.034,35.674,156.697
C09003=1052.825,218.119,-94.147,172.031,35.671,156.697
C09004=1052.819,217.870,-94.120,172.030,35.667,156.696
C09005=1052.813,217.622,-94.093,172.028,35.664,156.695
C09006=1052.806,217.373,-94.067,172.025,35.660,156.694
C09007=1052.800,217.125,-94.040,172.023,35.657,156.694
C09008=1052.793,216.876,-94.014,172.022,35.653,156.693
C09009=1052.787,216.628,-93.987,172.019,35.650,156.692
C09010=1052.781,216.380,-93.961,172.017,35.646,156.692
C09011=1052.775,216.131,-93.934,172.016,35.643,156.691
C09012=1052.769,215.882,-93.907,172.013,35.639,156.690
C09013=1052.762,215.634,-93.881,172.011,35.635,156.690
C09014=1052.756,215.385,-93.854,172.009,35.632,156.689
C09015=1052.749,215.137,-93.828,172.007,35.629,156.688
C09016=1052.743,214.888,-93.801,172.005,35.625,156.687
C09017=1052.736,214.640,-93.775,172.003,35.622,156.687
C09018=1052.730,214.391,-93.748,172.000,35.618,156.686
C09019=1052.724,214.143,-93.722,171.999,35.614,156.685
C09020=1052.718,213.895,-93.695,171.997,35.611,156.685
C09021=1052.711,213.645,-93.670,171.994,35.607,156.684
C09022=1052.705,213.397,-93.643,171.993,35.604,156.683
C09023=1052.699,213.148,-93.616,171.991,35.601,156.682
C09024=1052.692,212.900,-93.590,171.988,35.597,156.682
C09025=1052.687,212.651,-93.563,171.987,35.593,156.681
C09026=1052.680,212.403,-93.537,171.985,35.590,156.680
C09027=1052.674,212.154,-93.511,171.982,35.586,156.680
C09028=1052.667,211.906,-93.485,171.980,35.583,156.679
C09029=1052.661,211.658,-93.459,171.979,35.579,156.678
C09030=1052.655,211.408,-93.432,171.976,35.575,156.677
C09031=1052.648,211.160,-93.406,171.974,35.572,156.677
C09032=1052.642,210.912,-93.380,171.973,35.569,156.676
C09033=1052.635,210.663,-93.353,171.970,35.565,156.675
C09034=1052.629,210.415,-93.327,171.968,35.561,156.675
C09035=1052.623,210.166,-93.301,171.967,35.558,156.674
C09036=1052.617,209.918,-93.275,171.964,35.554,156.673
C09037=1052.610,209.669,-93.249,171.962,35.551,156.672
C09038=1052.604,209.420,-93.224,171.961,35.547,156.672
C09039=1052.598,209.172,-93.197,171.958,35.543,156.671
C09040=1052.591,208.923,-93.171,171.956,35.540,156.670
C09041=1052.585,208.674,-93.145,171.955,35.537,156.670
C09042=1052.579,208.428,-93.119,171.953,35.533,156.669
C09043=1052.572,208.183,-93.093,171.950,35.530,156.668
C09044=1052.565,207.937,-93.067,171.949,35.526,156.667
C09045=1052.560,207.691,-93.041,171.947,35.522,156.667
C09046=1052.553,207.445,-93.016,171.945,35.519,156.666
C09047=1052.547,207.200,-92.990,171.943,35.516,156.665
C09048=1052.540,206.953,-92.965,171.941,35.512,156.665
C09049=1052.534,206.707,-92.938,171.939,35.508,156.664
C09050=1052.509,205.656,-92.833,171.720,35.414,156.647
C09051=1052.503,205.407,-92.808,171.718,35.411,156.647
C09052=1052.496,205.158,-92.784,171.716,35.409,156.646
C09053=1052.490,204.909,-92.759,171.714,35.406,156.646
C09054=1052.485,204.661,-92.734,171.710,35.403,156.645
C09055=1052.479,204.412,-92.709,171.708,35.401,156.645
